KUKA KRL program: MyProgram_156().src

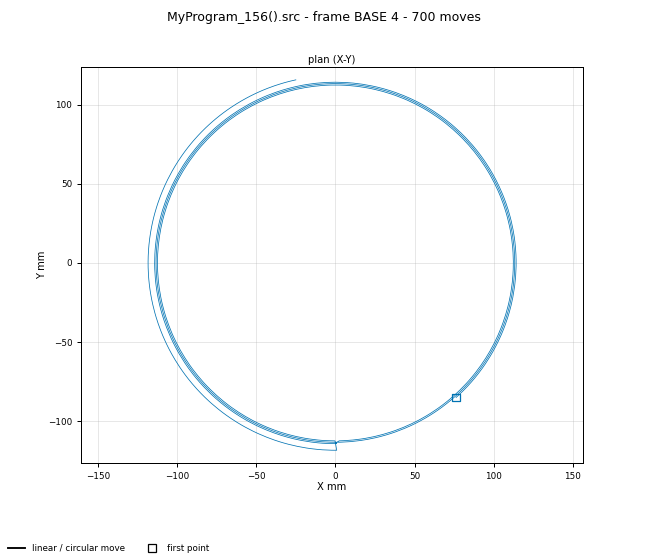
[picture p0: tool path of MyProgram_156().src in frame BASE 4, 700 of 700 moves have a stored position in this frame; points joined in program order, loops and branches not executed]
&ACCESS RVP
&REL 1
&PARAM TEMPLATE = C:\KRC\Roboter\Template\vorgabe
&PARAM EDITMASK = *
DEF MyProgram_156()
; ---- Setting reference (Base) ----
$BASE = BASE_DATA[4]

; --------------------------
; ---- Setting tool (TCP) ----
$TOOL = TOOL_DATA[3]
; --------------------------

$VEL.CP = VEL_APROX_PRINT
Startdeposition()
$VEL.CP = VEL_PRINT
LIN {X 76.2386,Y -85.0101,Z 120,A -51.5636,B 24.9513,C -1.613,E1 25.1077,E2 497.4724} C_DIS
LIN {X 78.7436,Y -82.698,Z 120,A -49.7889,B 24.9508,C -1.62,E1 25.1113,E2 495.6883} C_DIS
LIN {X 81.111,Y -80.3746,Z 120,A -48.1831,B 24.9508,C -1.6214,E1 25.1145,E2 494.086} C_DIS
LIN {X 83.3375,Y -78.0638,Z 120,A -46.5882,B 24.9505,C -1.6248,E1 25.1176,E2 492.4901} C_DIS
LIN {X 85.7956,Y -75.3542,Z 120,A -44.7139,B 24.9501,C -1.6313,E1 25.1211,E2 490.6088} C_DIS
LIN {X 88.0102,Y -72.7553,Z 120,A -42.9236,B 24.9496,C -1.6394,E1 25.1243,E2 488.8074} C_DIS
LIN {X 90.5109,Y -69.6191,Z 120,A -41.0242,B 24.9496,C -1.6396,E1 25.1275,E2 486.9167} C_DIS
LIN {X 92.7013,Y -66.6761,Z 120,A -39.1167,B 24.9491,C -1.6478,E1 25.1307,E2 484.999} C_DIS
LIN {X 94.7109,Y -63.7885,Z 120,A -37.4463,B 24.9491,C -1.6483,E1 25.1333,E2 483.3356} C_DIS
LIN {X 97.8312,Y -58.8925,Z 120,A -34.6127,B 24.9488,C -1.6529,E1 25.1375,E2 480.5054} C_DIS
LIN {X 99.5347,Y -55.9643,Z 120,A -32.8334,B 24.9483,C -1.6617,E1 25.14,E2 478.7147} C_DIS
LIN {X 101.2424,Y -52.813,Z 120,A -31.0463,B 24.948,C -1.6665,E1 25.1423,E2 476.9256} C_DIS
LIN {X 102.9812,Y -49.3349,Z 120,A -29.0203,B 24.9474,C -1.6759,E1 25.1448,E2 474.8882} C_DIS
LIN {X 104.7978,Y -45.3494,Z 120,A -26.7386,B 24.9467,C -1.6866,E1 25.1474,E2 472.5937} C_DIS
LIN {X 106.0833,Y -42.2573,Z 120,A -25.2084,B 24.9468,C -1.6848,E1 25.149,E2 471.0764} C_DIS
LIN {X 107.2709,Y -39.1408,Z 120,A -23.3343,B 24.9459,C -1.6995,E1 25.1509,E2 469.178} C_DIS
LIN {X 108.7458,Y -34.8355,Z 120,A -21.3851,B 24.9464,C -1.6909,E1 25.1525,E2 467.26} C_DIS
LIN {X 109.8552,Y -31.1591,Z 120,A -19.3865,B 24.9458,C -1.7005,E1 25.1541,E2 465.2504} C_DIS
LIN {X 111.0251,Y -26.6948,Z 120,A -17.1795,B 24.9457,C -1.7028,E1 25.1556,E2 463.0507} C_DIS
LIN {X 112.0611,Y -21.9428,Z 120,A -14.7665,B 24.9452,C -1.7094,E1 25.157,E2 460.6362} C_DIS
LIN {X 113.2585,Y -14.5453,Z 120,A -11.4137,B 24.9457,C -1.7024,E1 25.1585,E2 457.3196} C_DIS
LIN {X 113.8562,Y -8.7156,Z 120,A -7.9945,B 24.9436,C -1.7344,E1 25.1594,E2 453.8452} C_DIS
LIN {X 114.1732,Y -1.8883,Z 120,A -4.1574,B 24.9416,C -1.7648,E1 25.1598,E2 449.9591} C_DIS
LIN {X 114.1717,Y 1.9674,Z 120,A -2.7839,B 24.943,C -1.7446,E1 25.1598,E2 448.6415} C_DIS
LIN {X 114.0675,Y 5.2703,Z 120,A -0.544,B 24.9408,C -1.7775,E1 25.1595,E2 446.3374} C_DIS
LIN {X 113.8093,Y 9.3025,Z 120,A 1.5121,B 24.9403,C -1.7854,E1 25.159,E2 444.2749} C_DIS
LIN {X 113.3833,Y 13.5398,Z 120,A 2.9581,B 24.942,C -1.7596,E1 25.1586,E2 442.8981} C_DIS
LIN {X 112.9985,Y 16.4475,Z 120,A 5.1558,B 24.9394,C -1.7986,E1 25.1576,E2 440.6215} C_DIS
LIN {X 112.2633,Y 20.8817,Z 120,A 6.6108,B 24.9414,C -1.768,E1 25.157,E2 439.2473} C_DIS
LIN {X 111.1091,Y 26.3486,Z 120,A 9.4907,B 24.9406,C -1.7803,E1 25.1553,E2 436.355} C_DIS
LIN {X 110.4068,Y 29.1515,Z 120,A 10.964,B 24.9402,C -1.7859,E1 25.1542,E2 434.877} C_DIS
LIN {X 109.1219,Y 33.6376,Z 120,A 13.3219,B 24.9397,C -1.7938,E1 25.1524,E2 432.5139} C_DIS
LIN {X 108.0151,Y 37.0421,Z 120,A 15.1558,B 24.9392,C -1.801,E1 25.1507,E2 430.6734} C_DIS
LIN {X 106.7656,Y 40.4989,Z 120,A 16.8898,B 24.9392,C -1.8014,E1 25.149,E2 428.9482} C_DIS
LIN {X 105.6594,Y 43.3037,Z 120,A 18.5007,B 24.9386,C -1.8104,E1 25.1473,E2 427.3249} C_DIS
LIN {X 103.451,Y 48.3421,Z 120,A 21.0822,B 24.9386,C -1.81,E1 25.1444,E2 424.7583} C_DIS
LIN {X 101.3471,Y 52.6143,Z 120,A 23.6617,B 24.9375,C -1.8255,E1 25.1412,E2 422.156} C_DIS
LIN {X 99.5345,Y 55.9646,Z 120,A 25.5138,B 24.9374,C -1.8281,E1 25.1387,E2 420.3076} C_DIS
LIN {X 97.6359,Y 59.2139,Z 120,A 27.3716,B 24.9371,C -1.8317,E1 25.136,E2 418.4507} C_DIS
LIN {X 95.1175,Y 63.1811,Z 120,A 29.4198,B 24.9377,C -1.8236,E1 25.133,E2 416.4319} C_DIS
LIN {X 93.6732,Y 65.3024,Z 120,A 30.9566,B 24.9366,C -1.8384,E1 25.1305,E2 414.8677} C_DIS
LIN {X 91.5095,Y 68.302,Z 120,A 32.8457,B 24.9362,C -1.8446,E1 25.1273,E2 412.9732} C_DIS
LIN {X 89.4167,Y 71.0195,Z 120,A 35.121,B 24.9341,C -1.8744,E1 25.1233,E2 410.6381} C_DIS
LIN {X 86.5957,Y 74.4344,Z 120,A 36.6899,B 24.9359,C -1.8494,E1 25.1206,E2 409.1353} C_DIS
LIN {X 82.3085,Y 79.1477,Z 120,A 39.5817,B 24.9364,C -1.8427,E1 25.1152,E2 406.2722} C_DIS
LIN {X 79.422,Y 82.0442,Z 120,A 41.9376,B 24.9351,C -1.8609,E1 25.1104,E2 403.8831} C_DIS
LIN {X 75.0439,Y 86.0666,Z 120,A 44.8129,B 24.9351,C -1.8621,E1 25.1045,E2 401.0167} C_DIS
LIN {X 72.8834,Y 87.9037,Z 120,A 46.8965,B 24.9327,C -1.8949,E1 25.0999,E2 398.8635} C_DIS
LIN {X 69.624,Y 90.5071,Z 120,A 48.4215,B 24.9342,C -1.8729,E1 25.0967,E2 397.3962} C_DIS
LIN {X 66.4308,Y 92.8763,Z 120,A 50.5415,B 24.9336,C -1.882,E1 25.0918,E2 395.2621} C_DIS
LIN {X 62.5852,Y 95.5104,Z 120,A 52.7023,B 24.9339,C -1.8778,E1 25.0869,E2 393.1184} C_DIS
LIN {X 60.3508,Y 96.9374,Z 120,A 54.0595,B 24.9337,C -1.8811,E1 25.0837,E2 391.7578} C_DIS
LIN {X 57.0857,Y 98.8955,Z 120,A 55.9041,B 24.9337,C -1.8811,E1 25.0792,E2 389.9191} C_DIS
LIN {X 54.6498,Y 100.2621,Z 120,A 57.4025,B 24.9332,C -1.8873,E1 25.0755,E2 388.4101} C_DIS
LIN {X 51.2738,Y 102.0315,Z 120,A 59.4609,B 24.9326,C -1.8963,E1 25.0704,E2 386.3362} C_DIS
LIN {X 47.3144,Y 103.9259,Z 120,A 61.617,B 24.9326,C -1.8969,E1 25.0649,E2 384.1842} C_DIS
LIN {X 43.2541,Y 105.6796,Z 120,A 63.9554,B 24.932,C -1.9046,E1 25.0589,E2 381.833} C_DIS
LIN {X 38.0509,Y 107.6626,Z 120,A 66.4845,B 24.9326,C -1.8955,E1 25.0523,E2 379.3308} C_DIS
LIN {X 34.5457,Y 108.8395,Z 120,A 68.6595,B 24.9315,C -1.9111,E1 25.0465,E2 377.123} C_DIS
LIN {X 30.7609,Y 109.968,Z 120,A 70.3134,B 24.9325,C -1.898,E1 25.0421,E2 375.5027} C_DIS
LIN {X 26.7576,Y 111.0098,Z 120,A 72.2957,B 24.9327,C -1.8952,E1 25.0368,E2 373.5301} C_DIS
LIN {X 23.2459,Y 111.7978,Z 120,A 74.2356,B 24.9322,C -1.902,E1 25.0314,E2 371.5767} C_DIS
LIN {X 16.9448,Y 112.9255,Z 120,A 77.3058,B 24.9325,C -1.8969,E1 25.023,E2 368.5218} C_DIS
LIN {X 11.441,Y 113.6149,Z 120,A 80.939,B 24.9298,C -1.9344,E1 25.0127,E2 364.8022} C_DIS
LIN {X 6.4298,Y 114.0075,Z 120,A 82.3847,B 24.9332,C -1.8877,E1 25.009,E2 363.4678} C_DIS
LIN {X 0.0192,Y 114.1907,Z 120,A 85.9521,B 24.9322,C -1.9022,E1 24.999,E2 359.8666} C_DIS
LIN {X -5.4539,Y 114.0596,Z 120,A 88.5974,B 24.9325,C -1.897,E1 24.9916,E2 357.2332} C_DIS
LIN {X -12.2551,Y 113.5297,Z 120,A 91.9236,B 24.9329,C -1.8913,E1 24.9824,E2 353.9192} C_DIS
LIN {X -17.9444,Y 112.771,Z 120,A 94.876,B 24.9329,C -1.8924,E1 24.9742,E2 350.9618} C_DIS
LIN {X -21.0211,Y 112.2385,Z 120,A 97.068,B 24.931,C -1.9178,E1 24.968,E2 348.7072} C_DIS
LIN {X -24.9456,Y 111.4323,Z 120,A 98.8245,B 24.932,C -1.9052,E1 24.9633,E2 346.9784} C_DIS
LIN {X -29.9895,Y 110.1804,Z 120,A 101.1547,B 24.933,C -1.8909,E1 24.9571,E2 344.6789} C_DIS
LIN {X -33.4559,Y 109.1782,Z 120,A 103.0604,B 24.9328,C -1.8928,E1 24.9519,E2 342.7653} C_DIS
LIN {X -37.39,Y 107.8945,Z 120,A 105.1169,B 24.9331,C -1.8895,E1 24.9465,E2 340.713} C_DIS
LIN {X -42.6939,Y 105.9076,Z 120,A 108.1852,B 24.9327,C -1.8951,E1 24.9385,E2 337.6247} C_DIS
LIN {X -46.0433,Y 104.4952,Z 120,A 110.2515,B 24.9321,C -1.9025,E1 24.9331,E2 335.5359} C_DIS
LIN {X -49.5357,Y 102.8847,Z 120,A 111.373,B 24.9347,C -1.8658,E1 24.9305,E2 334.4987} C_DIS
LIN {X -51.8511,Y 101.7375,Z 120,A 112.8876,B 24.9343,C -1.8727,E1 24.9267,E2 332.9637} C_DIS
LIN {X -54.8258,Y 100.1667,Z 120,A 114.7339,B 24.934,C -1.8764,E1 24.9221,E2 331.1036} C_DIS
LIN {X -60.8098,Y 96.6506,Z 120,A 118.4997,B 24.9336,C -1.8816,E1 24.913,E2 327.3137} C_DIS
LIN {X -65.554,Y 93.4983,Z 120,A 121.5436,B 24.9335,C -1.8836,E1 24.906,E2 324.2548} C_DIS
LIN {X -68.6343,Y 91.26,Z 120,A 122.9574,B 24.9352,C -1.8591,E1 24.903,E2 322.8943} C_DIS
LIN {X -71.6379,Y 88.9222,Z 120,A 124.9947,B 24.9352,C -1.8602,E1 24.8985,E2 320.8468} C_DIS
LIN {X -74.5863,Y 86.4663,Z 120,A 126.8349,B 24.9357,C -1.8523,E1 24.8946,E2 319.0183} C_DIS
LIN {X -77.1405,Y 84.1926,Z 120,A 128.5557,B 24.9359,C -1.8486,E1 24.891,E2 317.2995} C_DIS
LIN {X -79.9011,Y 81.5787,Z 120,A 130.5038,B 24.9361,C -1.8456,E1 24.8871,E2 315.3503} C_DIS
LIN {X -82.3085,Y 79.1477,Z 120,A 132.1826,B 24.9365,C -1.8399,E1 24.8838,E2 313.678} C_DIS
LIN {X -85.738,Y 75.4202,Z 120,A 134.871,B 24.9365,C -1.8393,E1 24.8788,E2 310.9789} C_DIS
LIN {X -87.8307,Y 72.9712,Z 120,A 136.3419,B 24.9373,C -1.8292,E1 24.8762,E2 309.5253} C_DIS
LIN {X -92.1157,Y 67.4814,Z 120,A 139.6684,B 24.9384,C -1.813,E1 24.8706,E2 306.2217} C_DIS
LIN {X -94.7744,Y 63.6947,Z 120,A 142.1042,B 24.9385,C -1.8111,E1 24.8667,E2 303.7785} C_DIS
LIN {X -96.2133,Y 61.4987,Z 120,A 143.4703,B 24.9386,C -1.8093,E1 24.8646,E2 302.4098} C_DIS
LIN {X -99.3647,Y 56.2686,Z 120,A 146.8399,B 24.9384,C -1.8126,E1 24.8598,E2 299.0147} C_DIS
LIN {X -101.3602,Y 52.5893,Z 120,A 148.7275,B 24.9394,C -1.7978,E1 24.8573,E2 297.1523} C_DIS
LIN {X -103.3993,Y 48.4532,Z 120,A 151.1537,B 24.9396,C -1.7954,E1 24.8544,E2 294.7189} C_DIS
LIN {X -106.1097,Y 42.19,Z 120,A 154.3823,B 24.9408,C -1.777,E1 24.8509,E2 291.5163} C_DIS
LIN {X -107.202,Y 39.3297,Z 120,A 157.0353,B 24.9381,C -1.8172,E1 24.8483,E2 288.7523} C_DIS
LIN {X -109.0942,Y 33.727,Z 120,A 158.6626,B 24.9423,C -1.7539,E1 24.847,E2 287.2666} C_DIS
LIN {X -109.8654,Y 31.1231,Z 120,A 160.3997,B 24.9416,C -1.7645,E1 24.8456,E2 285.4943} C_DIS
LIN {X -111.222,Y 25.8599,Z 120,A 162.8599,B 24.9429,C -1.7451,E1 24.8439,E2 283.0659} C_DIS
LIN {X -111.7459,Y 23.4986,Z 120,A 164.4267,B 24.9423,C -1.7552,E1 24.843,E2 281.4659} C_DIS
LIN {X -112.3914,Y 20.1798,Z 120,A 166.0871,B 24.9427,C -1.7483,E1 24.8421,E2 279.812} C_DIS
LIN {X -113.0751,Y 15.9085,Z 120,A 168.2456,B 24.9432,C -1.7408,E1 24.8412,E2 277.6586} C_DIS
LIN {X -113.6182,Y 11.4094,Z 120,A 170.518,B 24.9437,C -1.7333,E1 24.8405,E2 275.3904} C_DIS
LIN {X -113.8778,Y 8.4455,Z 120,A 172.0471,B 24.9439,C -1.7299,E1 24.8401,E2 273.8604} C_DIS
LIN {X -114.0597,Y 5.4493,Z 120,A 173.7958,B 24.9436,C -1.7347,E1 24.8399,E2 272.0897} C_DIS
LIN {X -114.1877,Y -0.5465,Z 120,A 176.6355,B 24.9447,C -1.7181,E1 24.8399,E2 269.2724} C_DIS
LIN {X -114.1212,Y -3.9481,Z 120,A 178.4619,B 24.9447,C -1.7173,E1 24.8399,E2 267.4369} C_DIS
LIN {X -113.7849,Y -9.6066,Z 120,A -178.4365,B 24.9447,C -1.7185,E1 24.8406,E2 264.3139} C_DIS
LIN {X -113.4701,Y -12.7992,Z 120,A -177.3293,B 24.9463,C -1.6932,E1 24.8409,E2 263.2605} C_DIS
LIN {X -112.9768,Y -16.5995,Z 120,A -174.8603,B 24.9453,C -1.7089,E1 24.8419,E2 260.739} C_DIS
LIN {X -112.4554,Y -19.824,Z 120,A -173.585,B 24.9465,C -1.6891,E1 24.8425,E2 259.5035} C_DIS
LIN {X -111.8985,Y -22.7553,Z 120,A -172.0568,B 24.9468,C -1.6857,E1 24.8433,E2 257.9744} C_DIS
LIN {X -111.1311,Y -26.2534,Z 120,A -170.2104,B 24.947,C -1.682,E1 24.8444,E2 256.1259} C_DIS
LIN {X -110.272,Y -29.6503,Z 120,A -168.5105,B 24.9475,C -1.6743,E1 24.8456,E2 254.4346} C_DIS
LIN {X -109.3885,Y -32.761,Z 120,A -166.8336,B 24.9476,C -1.6715,E1 24.8469,E2 252.7546} C_DIS
LIN {X -108.25,Y -36.3455,Z 120,A -164.2457,B 24.9462,C -1.6942,E1 24.8493,E2 250.0977} C_DIS
LIN {X -106.6107,Y -40.9073,Z 120,A -162.5705,B 24.9486,C -1.6562,E1 24.8509,E2 248.5037} C_DIS
LIN {X -103.8533,Y -47.4753,Z 120,A -158.9719,B 24.9492,C -1.6467,E1 24.8548,E2 244.9078} C_DIS
LIN {X -102.3457,Y -50.6399,Z 120,A -157.1253,B 24.9492,C -1.6453,E1 24.8571,E2 243.0545} C_DIS
LIN {X -100.6772,Y -53.8846,Z 120,A -155.022,B 24.9489,C -1.6513,E1 24.8598,E2 240.9258} C_DIS
LIN {X -98.6721,Y -57.4745,Z 120,A -153.1831,B 24.9498,C -1.6366,E1 24.8624,E2 239.1125} C_DIS
LIN {X -95.0936,Y -63.2174,Z 120,A -149.9823,B 24.9508,C -1.6197,E1 24.8671,E2 235.9356} C_DIS
LIN {X -92.8073,Y -66.5275,Z 120,A -147.8552,B 24.9508,C -1.619,E1 24.8705,E2 233.7997} C_DIS
LIN {X -89.9271,Y -70.3736,Z 120,A -145.4098,B 24.9512,C -1.6144,E1 24.8746,E2 231.3534} C_DIS
LIN {X -87.8624,Y -72.9331,Z 120,A -143.7453,B 24.9514,C -1.6111,E1 24.8776,E2 229.6891} C_DIS
LIN {X -85.7278,Y -75.4319,Z 120,A -141.86,B 24.951,C -1.6171,E1 24.8811,E2 227.7812} C_DIS
LIN {X -82.7328,Y -78.7067,Z 120,A -139.6862,B 24.9514,C -1.6099,E1 24.8852,E2 225.6149} C_DIS
LIN {X -78.5953,Y -82.8376,Z 120,A -137.0135,B 24.9525,C -1.5929,E1 24.8905,E2 222.9715} C_DIS
LIN {X -75.4162,Y -85.7414,Z 120,A -134.6481,B 24.9522,C -1.597,E1 24.8954,E2 220.5867} C_DIS
LIN {X -72.2085,Y -88.4598,Z 120,A -132.6218,B 24.9527,C -1.5895,E1 24.8997,E2 218.5706} C_DIS
LIN {X -69.7896,Y -90.3796,Z 120,A -130.9737,B 24.9526,C -1.5908,E1 24.9034,E2 216.9133} C_DIS
LIN {X -66.8325,Y -92.5897,Z 120,A -129.0989,B 24.9527,C -1.5885,E1 24.9076,E2 215.0374} C_DIS
LIN {X -63.6085,Y -94.8328,Z 120,A -127.1457,B 24.953,C -1.5845,E1 24.9121,E2 213.0871} C_DIS
LIN {X -59.7782,Y -97.2921,Z 120,A -124.5248,B 24.9523,C -1.5953,E1 24.9184,E2 210.4323} C_DIS
LIN {X -57.0074,Y -98.9404,Z 120,A -123.3308,B 24.9535,C -1.575,E1 24.9212,E2 209.2829} C_DIS
LIN {X -54.373,Y -100.4123,Z 120,A -121.6249,B 24.9532,C -1.5811,E1 24.9254,E2 207.5577} C_DIS
LIN {X -50.3798,Y -102.4747,Z 120,A -119.524,B 24.9537,C -1.5717,E1 24.9306,E2 205.4736} C_DIS
LIN {X -48.1213,Y -103.5538,Z 120,A -118.2046,B 24.9537,C -1.5729,E1 24.9339,E2 204.148} C_DIS
LIN {X -43.8969,Y -105.4151,Z 120,A -115.5924,B 24.953,C -1.583,E1 24.9407,E2 201.5055} C_DIS
LIN {X -39.103,Y -107.2847,Z 120,A -113.2857,B 24.9539,C -1.5688,E1 24.9467,E2 199.2278} C_DIS
LIN {X -34.3136,Y -108.9123,Z 120,A -110.9186,B 24.9544,C -1.5594,E1 24.9529,E2 196.8787} C_DIS
LIN {X -30.0803,Y -110.1559,Z 120,A -108.525,B 24.9541,C -1.5657,E1 24.9594,E2 194.4664} C_DIS
LIN {X -26.125,Y -111.1607,Z 120,A -106.4824,B 24.9541,C -1.5643,E1 24.9649,E2 192.4242} C_DIS
LIN {X -21.571,Y -112.1327,Z 120,A -104.1706,B 24.9543,C -1.5622,E1 24.9712,E2 190.1146} C_DIS
LIN {X -15.0454,Y -113.1937,Z 120,A -100.3366,B 24.953,C -1.584,E1 24.982,E2 186.2258} C_DIS
LIN {X -11.092,Y -113.6502,Z 120,A -98.9589,B 24.9546,C -1.5565,E1 24.9856,E2 184.9123} C_DIS
LIN {X -8.1981,Y -113.895,Z 120,A -96.7306,B 24.9526,C -1.5905,E1 24.9921,E2 182.6025} C_DIS
LIN {X -3.6609,Y -114.13,Z 120,A -94.4111,B 24.9525,C -1.5926,E1 24.9985,E2 180.2778} C_DIS
LIN {X 0.826,Y -114.1802,Z 120,A -94.2003,B 24.9576,C -1.5037,E1 24.9986,E2 180.2778} C_DIS
Enddeposition()
LIN {X 0.826,Y -114.1802,Z 120,A -94.2003,B 24.9576,C -1.5037,E1 24.9986,E2 180.2778} C_DIS
Startdeposition()
$VEL.CP = VEL_PRINT
LIN {X 0.5604,Y -113.3011,Z 120,A -94.2192,B 24.9565,C -1.5242,E1 24.9986,E2 180.248} C_DIS
LIN {X -3.0264,Y -113.2628,Z 120,A -96.4904,B 24.9576,C -1.5045,E1 24.9922,E2 182.5661} C_DIS
LIN {X -8.552,Y -112.9802,Z 120,A -98.2379,B 24.955,C -1.5491,E1 24.9876,E2 184.2085} C_DIS
LIN {X -14.2204,Y -112.407,Z 120,A -101.0574,B 24.9549,C -1.552,E1 24.9798,E2 187.0228} C_DIS
LIN {X -17.25,Y -111.9816,Z 120,A -102.8667,B 24.9555,C -1.5412,E1 24.9747,E2 188.8592} C_DIS
LIN {X -20.5468,Y -111.4249,Z 120,A -104.7709,B 24.956,C -1.5328,E1 24.9694,E2 190.7855} C_DIS
LIN {X -25.1163,Y -110.4842,Z 120,A -106.6838,B 24.9548,C -1.5527,E1 24.9643,E2 192.6533} C_DIS
LIN {X -27.1879,Y -109.9926,Z 120,A -108.0573,B 24.9555,C -1.5408,E1 24.9605,E2 194.0571} C_DIS
LIN {X -30.4687,Y -109.1296,Z 120,A -109.4981,B 24.9548,C -1.5534,E1 24.9567,E2 195.4701} C_DIS
LIN {X -32.6296,Y -108.5031,Z 120,A -110.7626,B 24.9551,C -1.5489,E1 24.9532,E2 196.7475} C_DIS
LIN {X -36.2392,Y -107.3506,Z 120,A -112.7597,B 24.9551,C -1.547,E1 24.9479,E2 198.7526} C_DIS
LIN {X -40.1007,Y -105.9687,Z 120,A -115.9071,B 24.9576,C -1.5046,E1 24.9394,E2 202.0074} C_DIS
LIN {X -46.0582,Y -103.5199,Z 120,A -117.9469,B 24.9545,C -1.5582,E1 24.9345,E2 203.9245} C_DIS
LIN {X -49.2376,Y -102.0447,Z 120,A -119.94,B 24.9549,C -1.5511,E1 24.9294,E2 205.9395} C_DIS
LIN {X -52.2376,Y -100.5438,Z 120,A -121.7297,B 24.955,C -1.5494,E1 24.9249,E2 207.7381} C_DIS
LIN {X -56.2111,Y -98.3759,Z 120,A -125.0629,B 24.9573,C -1.5102,E1 24.9166,E2 211.1743} C_DIS
LIN {X -62.0967,Y -94.7709,Z 120,A -127.6485,B 24.9549,C -1.5522,E1 24.9108,E2 213.6683} C_DIS
LIN {X -65.4261,Y -92.5044,Z 120,A -129.2346,B 24.9536,C -1.574,E1 24.9072,E2 215.2079} C_DIS
LIN {X -67.4604,Y -91.0326,Z 120,A -130.8072,B 24.9542,C -1.5639,E1 24.9036,E2 216.8103} C_DIS
LIN {X -70.3716,Y -88.7991,Z 120,A -132.4081,B 24.9534,C -1.5776,E1 24.9001,E2 218.3844} C_DIS
LIN {X -72.4498,Y -87.1118,Z 120,A -133.9467,B 24.9537,C -1.5727,E1 24.8968,E2 219.9406} C_DIS
LIN {X -75.6065,Y -84.3865,Z 120,A -136.0737,B 24.9535,C -1.5761,E1 24.8923,E2 222.0677} C_DIS
LIN {X -79.0329,Y -81.1884,Z 120,A -138.5976,B 24.9535,C -1.5748,E1 24.8872,E2 224.6052} C_DIS
LIN {X -82.1695,Y -78.0121,Z 120,A -140.6064,B 24.9526,C -1.5897,E1 24.8833,E2 226.587} C_DIS
LIN {X -84.1808,Y -75.8363,Z 120,A -142.2397,B 24.9528,C -1.5877,E1 24.8802,E2 228.2325} C_DIS
LIN {X -86.4828,Y -73.2003,Z 120,A -144.0611,B 24.9526,C -1.5897,E1 24.8769,E2 230.0573} C_DIS
LIN {X -88.8268,Y -70.3366,Z 120,A -145.8907,B 24.9523,C -1.5959,E1 24.8737,E2 231.8808} C_DIS
LIN {X -91.1598,Y -67.2868,Z 120,A -147.7112,B 24.9517,C -1.6055,E1 24.8707,E2 233.6871} C_DIS
LIN {X -92.9577,Y -64.7789,Z 120,A -149.2891,B 24.9515,C -1.6088,E1 24.8681,E2 235.265} C_DIS
LIN {X -94.2783,Y -62.8439,Z 120,A -151.1301,B 24.9529,C -1.5858,E1 24.8652,E2 237.1699} C_DIS
LIN {X -96.5397,Y -59.3112,Z 120,A -152.7773,B 24.9514,C -1.6101,E1 24.8629,E2 238.7677} C_DIS
LIN {X -97.9455,Y -56.9602,Z 120,A -154.4851,B 24.952,C -1.6011,E1 24.8604,E2 240.5058} C_DIS
LIN {X -99.5879,Y -54.034,Z 120,A -155.8188,B 24.9508,C -1.6201,E1 24.8587,E2 241.8013} C_DIS
LIN {X -101.1826,Y -50.9895,Z 120,A -157.5902,B 24.9506,C -1.6236,E1 24.8564,E2 243.5738} C_DIS
LIN {X -102.5679,Y -48.1393,Z 120,A -158.9446,B 24.9497,C -1.638,E1 24.8548,E2 244.9012} C_DIS
LIN {X -104.4003,Y -44.0227,Z 120,A -161.4285,B 24.9498,C -1.6364,E1 24.852,E2 247.4024} C_DIS
LIN {X -105.7208,Y -40.7553,Z 120,A -163.1504,B 24.9494,C -1.644,E1 24.8502,E2 249.1159} C_DIS
LIN {X -107.2805,Y -36.4471,Z 120,A -165.3923,B 24.9487,C -1.6539,E1 24.8482,E2 251.3469} C_DIS
LIN {X -107.9978,Y -34.2683,Z 120,A -166.8507,B 24.9493,C -1.6457,E1 24.8469,E2 252.8334} C_DIS
LIN {X -109.0319,Y -30.8136,Z 120,A -168.5498,B 24.9486,C -1.6562,E1 24.8456,E2 254.5172} C_DIS
LIN {X -109.9863,Y -27.2134,Z 120,A -170.2804,B 24.9479,C -1.668,E1 24.8444,E2 256.2298} C_DIS
LIN {X -110.5155,Y -24.9808,Z 120,A -171.7509,B 24.9484,C -1.6594,E1 24.8434,E2 257.7293} C_DIS
LIN {X -111.2888,Y -21.2665,Z 120,A -173.5467,B 24.9477,C -1.6703,E1 24.8424,E2 259.5098} C_DIS
LIN {X -111.883,Y -17.8876,Z 120,A -175.4201,B 24.9477,C -1.6703,E1 24.8416,E2 261.3942} C_DIS
LIN {X -112.4605,Y -13.8002,Z 120,A -177.5051,B 24.9473,C -1.6771,E1 24.8408,E2 263.4756} C_DIS
LIN {X -112.8326,Y -10.3075,Z 120,A -179.2013,B 24.9467,C -1.686,E1 24.8404,E2 265.1608} C_DIS
LIN {X -113.1095,Y -6.618,Z 120,A 179.1384,B 24.9458,C -1.7002,E1 24.84,E2 266.7971} C_DIS
LIN {X -113.247,Y -3.543,Z 120,A 177.6963,B 24.9452,C -1.7097,E1 24.8399,E2 268.2252} C_DIS
LIN {X -113.3003,Y -0.7681,Z 120,A 175.9113,B 24.9459,C -1.6994,E1 24.8398,E2 270.0456} C_DIS
LIN {X -113.2699,Y 2.7974,Z 120,A 174.1791,B 24.9453,C -1.708,E1 24.8398,E2 271.7677} C_DIS
LIN {X -113.1305,Y 6.2384,Z 120,A 172.3105,B 24.9453,C -1.7087,E1 24.8401,E2 273.6459} C_DIS
LIN {X -112.8168,Y 10.4788,Z 120,A 170.1496,B 24.9449,C -1.7153,E1 24.8406,E2 275.804} C_DIS
LIN {X -112.4248,Y 14.0825,Z 120,A 168.3044,B 24.9445,C -1.7208,E1 24.8412,E2 277.6472} C_DIS
LIN {X -111.9397,Y 17.5208,Z 120,A 166.5565,B 24.9441,C -1.7268,E1 24.8419,E2 279.3911} C_DIS
LIN {X -111.3768,Y 20.8095,Z 120,A 164.8263,B 24.9439,C -1.7306,E1 24.8428,E2 281.1226} C_DIS
LIN {X -110.7164,Y 24.0691,Z 120,A 163.1268,B 24.9436,C -1.7353,E1 24.8438,E2 282.8208} C_DIS
LIN {X -109.9826,Y 27.2287,Z 120,A 161.4836,B 24.9432,C -1.7405,E1 24.8448,E2 284.4613} C_DIS
LIN {X -109.0539,Y 30.736,Z 120,A 159.6851,B 24.9428,C -1.7477,E1 24.8461,E2 286.253} C_DIS
LIN {X -108.3381,Y 33.1728,Z 120,A 158.0515,B 24.9434,C -1.7383,E1 24.8475,E2 287.9186} C_DIS
LIN {X -106.831,Y 37.7443,Z 120,A 156.0026,B 24.9419,C -1.7609,E1 24.8493,E2 289.9253} C_DIS
LIN {X -105.7069,Y 40.7913,Z 120,A 154.2658,B 24.9418,C -1.7623,E1 24.851,E2 291.6686} C_DIS
LIN {X -104.4838,Y 43.8246,Z 120,A 152.4811,B 24.9418,C -1.7623,E1 24.8529,E2 293.4631} C_DIS
LIN {X -103.0723,Y 47.0513,Z 120,A 150.6971,B 24.9414,C -1.7676,E1 24.855,E2 295.2443} C_DIS
LIN {X -101.2371,Y 50.8809,Z 120,A 148.7442,B 24.9405,C -1.7816,E1 24.8573,E2 297.1742} C_DIS
LIN {X -98.9316,Y 55.2266,Z 120,A 146.2901,B 24.9399,C -1.7903,E1 24.8606,E2 299.6206} C_DIS
LIN {X -97.2506,Y 58.1383,Z 120,A 144.5048,B 24.9399,C -1.7919,E1 24.8631,E2 301.4115} C_DIS
LIN {X -95.4464,Y 61.0528,Z 120,A 142.9799,B 24.9389,C -1.8051,E1 24.8653,E2 302.9127} C_DIS
LIN {X -93.7931,Y 63.5632,Z 120,A 141.4771,B 24.9386,C -1.81,E1 24.8676,E2 304.4112} C_DIS
LIN {X -92.0085,Y 66.1211,Z 120,A 138.7674,B 24.9413,C -1.7701,E1 24.8722,E2 307.2292} C_DIS
LIN {X -88.8362,Y 70.3247,Z 120,A 136.8806,B 24.9388,C -1.8075,E1 24.8753,E2 309.0358} C_DIS
LIN {X -87.2193,Y 72.3204,Z 120,A 134.6491,B 24.941,C -1.7745,E1 24.8795,E2 311.3561} C_DIS
LIN {X -83.3552,Y 76.7422,Z 120,A 132.6535,B 24.9379,C -1.8201,E1 24.883,E2 313.252} C_DIS
LIN {X -80.9831,Y 79.243,Z 120,A 130.8101,B 24.9379,C -1.8205,E1 24.8866,E2 315.1026} C_DIS
LIN {X -78.498,Y 81.7039,Z 120,A 129.0384,B 24.9376,C -1.8246,E1 24.8901,E2 316.8717} C_DIS
LIN {X -75.7216,Y 84.2835,Z 120,A 127.1635,B 24.9372,C -1.8308,E1 24.894,E2 318.7397} C_DIS
LIN {X -71.4959,Y 87.8966,Z 120,A 124.3506,B 24.9367,C -1.837,E1 24.9,E2 321.5485} C_DIS
LIN {X -69.2532,Y 89.674,Z 120,A 122.1825,B 24.9385,C -1.8116,E1 24.905,E2 323.7851} C_DIS
LIN {X -65.3735,Y 92.542,Z 120,A 120.3391,B 24.9365,C -1.8402,E1 24.909,E2 325.5668} C_DIS
LIN {X -62.2386,Y 94.6774,Z 120,A 118.4668,B 24.9361,C -1.8458,E1 24.9133,E2 327.4319} C_DIS
LIN {X -59.3315,Y 96.5274,Z 120,A 116.8942,B 24.9354,C -1.8559,E1 24.917,E2 328.9855} C_DIS
LIN {X -56.5573,Y 98.177,Z 120,A 115.3408,B 24.935,C -1.8621,E1 24.9207,E2 330.5289} C_DIS
LIN {X -54.7472,Y 99.1993,Z 120,A 114.0842,B 24.9355,C -1.8556,E1 24.9238,E2 331.8045} C_DIS
LIN {X -51.81,Y 100.7632,Z 120,A 112.5543,B 24.9348,C -1.8646,E1 24.9276,E2 333.3172} C_DIS
LIN {X -49.6816,Y 101.8314,Z 120,A 111.2532,B 24.935,C -1.8626,E1 24.9308,E2 334.6265} C_DIS
LIN {X -47.0272,Y 103.0832,Z 120,A 109.6426,B 24.9352,C -1.8598,E1 24.9349,E2 336.2478} C_DIS
LIN {X -39.4582,Y 106.2117,Z 120,A 105.4481,B 24.9349,C -1.8634,E1 24.9458,E2 340.443} C_DIS
LIN {X -35.3941,Y 107.6335,Z 120,A 103.4893,B 24.9341,C -1.875,E1 24.9509,E2 342.3779} C_DIS
LIN {X -32.4048,Y 108.5697,Z 120,A 101.8356,B 24.9341,C -1.874,E1 24.9553,E2 344.0369} C_DIS
LIN {X -29.9852,Y 109.2635,Z 120,A 100.4488,B 24.9344,C -1.8707,E1 24.9591,E2 345.4338} C_DIS
LIN {X -24.1725,Y 110.6938,Z 120,A 97.469,B 24.9341,C -1.8755,E1 24.9672,E2 348.4062} C_DIS
LIN {X -20.8431,Y 111.3703,Z 120,A 95.6718,B 24.9341,C -1.8736,E1 24.9721,E2 350.2099} C_DIS
LIN {X -17.223,Y 111.9857,Z 120,A 93.6869,B 24.9345,C -1.8697,E1 24.9776,E2 352.2059} C_DIS
LIN {X -13.137,Y 112.5382,Z 120,A 92.0604,B 24.933,C -1.89,E1 24.982,E2 353.7855} C_DIS
LIN {X -9.4968,Y 112.9046,Z 120,A 89.7902,B 24.9342,C -1.8734,E1 24.9884,E2 356.0962} C_DIS
LIN {X -5.3758,Y 113.1759,Z 120,A 87.9936,B 24.9333,C -1.8863,E1 24.9933,E2 357.8625} C_DIS
LIN {X -1.9417,Y 113.2858,Z 120,A 85.9388,B 24.9342,C -1.8736,E1 24.9992,E2 359.948} C_DIS
LIN {X 2.8159,Y 113.2693,Z 120,A 83.6547,B 24.9338,C -1.879,E1 25.0055,E2 362.2188} C_DIS
LIN {X 6.0324,Y 113.1419,Z 120,A 81.6682,B 24.9349,C -1.864,E1 25.0111,E2 364.2402} C_DIS
LIN {X 9.4876,Y 112.9053,Z 120,A 80.0728,B 24.9344,C -1.8704,E1 25.0155,E2 365.8195} C_DIS
LIN {X 13.9176,Y 112.4462,Z 120,A 78.1496,B 24.9335,C -1.8839,E1 25.0208,E2 367.7094} C_DIS
LIN {X 16.6582,Y 112.0731,Z 120,A 76.7205,B 24.9335,C -1.8823,E1 25.0247,E2 369.1411} C_DIS
LIN {X 20.2987,Y 111.4695,Z 120,A 74.7508,B 24.9339,C -1.8772,E1 25.0302,E2 371.1207} C_DIS
LIN {X 23.2543,Y 110.8914,Z 120,A 73.3673,B 24.9336,C -1.8825,E1 25.0339,E2 372.4901} C_DIS
LIN {X 26.0046,Y 110.279,Z 120,A 71.8343,B 24.9339,C -1.8771,E1 25.0381,E2 374.0337} C_DIS
LIN {X 28.833,Y 109.5742,Z 120,A 70.4579,B 24.9337,C -1.8803,E1 25.0418,E2 375.4004} C_DIS
LIN {X 31.0593,Y 108.9623,Z 120,A 69.3581,B 24.9336,C -1.8825,E1 25.0448,E2 376.4933} C_DIS
LIN {X 33.5937,Y 108.2076,Z 120,A 67.8357,B 24.9342,C -1.8735,E1 25.0489,E2 378.0343} C_DIS
LIN {X 37.3046,Y 106.9852,Z 120,A 65.0288,B 24.9368,C -1.8362,E1 25.0565,E2 380.9238} C_DIS
LIN {X 42.4877,Y 105.0347,Z 120,A 63.1176,B 24.9343,C -1.8715,E1 25.0613,E2 382.7472} C_DIS
LIN {X 45.8341,Y 103.6197,Z 120,A 61.1747,B 24.9348,C -1.8649,E1 25.0663,E2 384.7012} C_DIS
LIN {X 49.3579,Y 101.9869,Z 120,A 59.2041,B 24.935,C -1.8622,E1 25.0712,E2 386.6729} C_DIS
LIN {X 52.8569,Y 100.2177,Z 120,A 57.3545,B 24.9348,C -1.8654,E1 25.0758,E2 388.5098} C_DIS
LIN {X 55.6354,Y 98.7033,Z 120,A 55.4893,B 24.9357,C -1.8516,E1 25.0804,E2 390.4022} C_DIS
LIN {X 59.8289,Y 96.2184,Z 120,A 53.2606,B 24.9353,C -1.8582,E1 25.0857,E2 392.6084} C_DIS
LIN {X 63.1587,Y 94.067,Z 120,A 51.482,B 24.9348,C -1.8649,E1 25.0898,E2 394.3652} C_DIS
LIN {X 65.5829,Y 92.3926,Z 120,A 49.7885,B 24.9356,C -1.8534,E1 25.0937,E2 396.0801} C_DIS
LIN {X 68.8412,Y 89.9915,Z 120,A 47.6174,B 24.9362,C -1.8442,E1 25.0986,E2 398.265} C_DIS
LIN {X 72.142,Y 87.3675,Z 120,A 45.6115,B 24.9362,C -1.8458,E1 25.1029,E2 400.2597} C_DIS
LIN {X 74.8577,Y 85.0526,Z 120,A 43.9915,B 24.9358,C -1.8504,E1 25.1063,E2 401.8624} C_DIS
LIN {X 77.0541,Y 83.0691,Z 120,A 42.332,B 24.9365,C -1.8401,E1 25.1097,E2 403.5396} C_DIS
LIN {X 79.532,Y 80.6976,Z 120,A 40.6274,B 24.9367,C -1.8378,E1 25.1132,E2 405.2426} C_DIS
LIN {X 81.3864,Y 78.8273,Z 120,A 39.1968,B 24.9372,C -1.8304,E1 25.116,E2 406.6844} C_DIS
LIN {X 84.3127,Y 75.689,Z 120,A 37.1583,B 24.9372,C -1.8314,E1 25.1198,E2 408.7116} C_DIS
LIN {X 86.7423,Y 72.8944,Z 120,A 35.0635,B 24.9381,C -1.8171,E1 25.1236,E2 410.8308} C_DIS
LIN {X 89.7885,Y 69.1047,Z 120,A 32.8258,B 24.9378,C -1.821,E1 25.1275,E2 413.0486} C_DIS
LIN {X 91.8285,Y 66.3735,Z 120,A 31.0737,B 24.9382,C -1.8154,E1 25.1304,E2 414.8055} C_DIS
LIN {X 93.3892,Y 64.1582,Z 120,A 29.6522,B 24.9386,C -1.8096,E1 25.1327,E2 416.2337} C_DIS
LIN {X 95.0391,Y 61.6873,Z 120,A 28.2026,B 24.9387,C -1.808,E1 25.1349,E2 417.6797} C_DIS
LIN {X 96.8528,Y 58.796,Z 120,A 26.5912,B 24.9387,C -1.8087,E1 25.1372,E2 419.2815} C_DIS
LIN {X 98.67,Y 55.6949,Z 120,A 24.8093,B 24.9389,C -1.8053,E1 25.1397,E2 421.062} C_DIS
LIN {X 99.9936,Y 53.2823,Z 120,A 23.2783,B 24.9396,C -1.7951,E1 25.1417,E2 422.6091} C_DIS
LIN {X 101.6033,Y 50.1421,Z 120,A 21.6178,B 24.9396,C -1.7958,E1 25.1438,E2 424.2592} C_DIS
LIN {X 103.0486,Y 47.104,Z 120,A 19.694,B 24.9406,C -1.7808,E1 25.1461,E2 426.2081} C_DIS
LIN {X 104.8701,Y 42.892,Z 120,A 17.6221,B 24.9403,C -1.7853,E1 25.1483,E2 428.2578} C_DIS
LIN {X 105.9094,Y 40.2572,Z 120,A 16.3196,B 24.9401,C -1.787,E1 25.1496,E2 429.5491} C_DIS
LIN {X 106.7088,Y 38.0925,Z 120,A 15.1167,B 24.9405,C -1.7818,E1 25.1508,E2 430.7574} C_DIS
LIN {X 107.7211,Y 35.1234,Z 120,A 13.4363,B 24.9411,C -1.7728,E1 25.1523,E2 432.4497} C_DIS
LIN {X 108.8089,Y 31.5987,Z 120,A 11.425,B 24.9419,C -1.7604,E1 25.1539,E2 434.4789} C_DIS
LIN {X 109.9078,Y 27.535,Z 120,A 9.323,B 24.9423,C -1.755,E1 25.1554,E2 436.5814} C_DIS
LIN {X 110.8666,Y 23.3751,Z 120,A 7.2529,B 24.9425,C -1.7523,E1 25.1566,E2 438.6458} C_DIS
LIN {X 112.0003,Y 17.1287,Z 120,A 4.025,B 24.9432,C -1.7413,E1 25.1582,E2 441.8806} C_DIS
LIN {X 112.9074,Y 9.4628,Z 120,A -0.5243,B 24.9459,C -1.6993,E1 25.1595,E2 446.502} C_DIS
LIN {X 113.22,Y 4.3507,Z 120,A -2.2496,B 24.9439,C -1.7304,E1 25.1597,E2 448.1438} C_DIS
LIN {X 113.3022,Y 0.3158,Z 120,A -4.4655,B 24.9448,C -1.7157,E1 25.1597,E2 450.3811} C_DIS
LIN {X 113.2156,Y -4.426,Z 120,A -7.0756,B 24.946,C -1.6982,E1 25.1596,E2 453.017} C_DIS
LIN {X 113.0427,Y -7.6661,Z 120,A -8.4016,B 24.9454,C -1.7073,E1 25.1593,E2 454.3137} C_DIS
LIN {X 112.4375,Y -13.9845,Z 120,A -12.2421,B 24.9479,C -1.6679,E1 25.1581,E2 458.2242} C_DIS
LIN {X 111.7615,Y -18.6224,Z 120,A -13.9413,B 24.9464,C -1.691,E1 25.1574,E2 459.8592} C_DIS
LIN {X 111.2061,Y -21.6957,Z 120,A -15.6698,B 24.9472,C -1.679,E1 25.1565,E2 461.6059} C_DIS
LIN {X 110.2591,Y -26.0909,Z 120,A -17.8774,B 24.9474,C -1.6746,E1 25.1551,E2 463.8109} C_DIS
LIN {X 109.4464,Y -29.3084,Z 120,A -19.3868,B 24.9473,C -1.677,E1 25.1541,E2 465.3059} C_DIS
LIN {X 108.5351,Y -32.5217,Z 120,A -20.9582,B 24.9473,C -1.677,E1 25.1529,E2 466.8683} C_DIS
LIN {X 107.5356,Y -35.6906,Z 120,A -22.8284,B 24.9482,C -1.663,E1 25.1512,E2 468.761} C_DIS
LIN {X 106.135,Y -39.6615,Z 120,A -24.9089,B 24.9485,C -1.6586,E1 25.1493,E2 470.8404} C_DIS
LIN {X 105.0867,Y -42.36,Z 120,A -26.9479,B 24.9504,C -1.6277,E1 25.1471,E2 472.9408} C_DIS
LIN {X 103.3309,Y -46.4774,Z 120,A -28.2046,B 24.9479,C -1.6669,E1 25.1458,E2 474.0982} C_DIS
LIN {X 101.845,Y -49.6532,Z 120,A -30.4248,B 24.9495,C -1.6409,E1 25.1431,E2 476.3679} C_DIS
LIN {X 100.5143,Y -52.2936,Z 120,A -31.9101,B 24.9498,C -1.6368,E1 25.1411,E2 477.8548} C_DIS
LIN {X 98.6195,Y -55.7854,Z 120,A -33.8833,B 24.9501,C -1.6325,E1 25.1385,E2 479.8279} C_DIS
LIN {X 96.638,Y -59.1494,Z 120,A -36.1161,B 24.9511,C -1.615,E1 25.1352,E2 482.0906} C_DIS
LIN {X 94.877,Y -61.9359,Z 120,A -37.4811,B 24.9506,C -1.624,E1 25.1332,E2 483.4276} C_DIS
LIN {X 92.9544,Y -64.7837,Z 120,A -39.0701,B 24.9505,C -1.6259,E1 25.1307,E2 485.0042} C_DIS
LIN {X 90.967,Y -67.5487,Z 120,A -40.9651,B 24.9512,C -1.6132,E1 25.1275,E2 486.92} C_DIS
LIN {X 88.4428,Y -70.8219,Z 120,A -43.038,B 24.9515,C -1.6084,E1 25.1239,E2 488.9946} C_DIS
LIN {X 86.2625,Y -73.4589,Z 120,A -44.6369,B 24.9515,C -1.6098,E1 25.1211,E2 490.5829} C_DIS
LIN {X 84.029,Y -76.0059,Z 120,A -46.3879,B 24.9518,C -1.6036,E1 25.1178,E2 492.3405} C_DIS
LIN {X 81.6477,Y -78.5563,Z 120,A -48.1508,B 24.9521,C -1.5993,E1 25.1144,E2 494.1061} C_DIS
LIN {X 78.7974,Y -81.4154,Z 120,A -50.1451,B 24.9522,C -1.5964,E1 25.1105,E2 496.0988} C_DIS
LIN {X 76.429,Y -83.6426,Z 120,A -51.8313,B 24.9526,C -1.5906,E1 25.107,E2 497.7918} C_DIS
LIN {X 73.6162,Y -86.1285,Z 120,A -53.6759,B 24.9527,C -1.5886,E1 25.1031,E2 499.6339} C_DIS
LIN {X 70.8265,Y -88.4391,Z 120,A -55.6447,B 24.9533,C -1.5783,E1 25.0988,E2 501.6194} C_DIS
LIN {X 67.4866,Y -91.0135,Z 120,A -57.6926,B 24.9533,C -1.5775,E1 25.0943,E2 503.6618} C_DIS
LIN {X 65.085,Y -92.7449,Z 120,A -58.9488,B 24.9529,C -1.5853,E1 25.0915,E2 504.8953} C_DIS
LIN {X 62.4445,Y -94.5416,Z 120,A -60.6389,B 24.9533,C -1.5787,E1 25.0875,E2 506.5954} C_DIS
LIN {X 59.828,Y -96.219,Z 120,A -62.3025,B 24.9537,C -1.5715,E1 25.0836,E2 508.2706} C_DIS
LIN {X 56.9388,Y -97.9578,Z 120,A -63.8474,B 24.9535,C -1.5755,E1 25.0799,E2 509.8012} C_DIS
LIN {X 53.5144,Y -99.8697,Z 120,A -65.8837,B 24.9538,C -1.5696,E1 25.0749,E2 511.8456} C_DIS
LIN {X 50.785,Y -101.2847,Z 120,A -67.5519,B 24.9543,C -1.5619,E1 25.0707,E2 513.5273} C_DIS
LIN {X 47.566,Y -102.8347,Z 120,A -69.8764,B 24.9558,C -1.5362,E1 25.0647,E2 515.9069} C_DIS
LIN {X 43.7161,Y -104.5296,Z 120,A -71.5185,B 24.9547,C -1.5544,E1 25.0606,E2 517.502} C_DIS
LIN {X 40.2572,Y -105.9094,Z 120,A -73.1492,B 24.9542,C -1.5629,E1 25.0564,E2 519.1088} C_DIS
LIN {X 38.0925,Y -106.7088,Z 120,A -74.5609,B 24.955,C -1.5505,E1 25.0526,E2 520.547} C_DIS
LIN {X 34.8025,Y -107.825,Z 120,A -76.0428,B 24.9544,C -1.5605,E1 25.0488,E2 522.0024} C_DIS
LIN {X 31.8433,Y -108.7363,Z 120,A -77.733,B 24.9548,C -1.5532,E1 25.0442,E2 523.7069} C_DIS
LIN {X 28.2679,Y -109.7195,Z 120,A -79.7081,B 24.9552,C -1.5468,E1 25.0389,E2 525.694} C_DIS
LIN {X 25.126,Y -110.4819,Z 120,A -81.2737,B 24.9551,C -1.5483,E1 25.0346,E2 527.254} C_DIS
LIN {X 20.3647,Y -111.4576,Z 120,A -83.9861,B 24.9559,C -1.5351,E1 25.0271,E2 529.9944} C_DIS
LIN {X 15.9244,Y -112.1777,Z 120,A -85.7023,B 24.9545,C -1.5578,E1 25.0225,E2 531.6552} C_DIS
LIN {X 9.4896,Y -112.9052,Z 120,A -89.1004,B 24.955,C -1.5504,E1 25.0131,E2 535.0684} C_DIS
LIN {X 3.3835,Y -113.2519,Z 120,A -92.1276,B 24.9549,C -1.5519,E1 25.0047,E2 538.0909} C_DIS
LIN {X 0.8144,Y -113.2977,Z 120,A -92.9638,B 24.9537,C -1.5717,E1 25.0025,E2 538.8801} C_DIS
Enddeposition()
LIN {X 0.8144,Y -113.2977,Z 120,A -92.9638,B 24.9537,C -1.5717,E1 25.0025,E2 538.8801} C_DIS
Startdeposition()
$VEL.CP = VEL_PRINT
LIN {X 2.4378,Y -112.3903,Z 120,A -92.1544,B 24.9528,C -1.5865,E1 25.0048,E2 538.0358} C_DIS
LIN {X 5.49,Y -112.284,Z 120,A -90.6058,B 24.9528,C -1.5867,E1 25.0091,E2 536.4872} C_DIS
LIN {X 8.1952,Y -112.1187,Z 120,A -89.2283,B 24.9528,C -1.5871,E1 25.013,E2 535.1092} C_DIS
LIN {X 10.9817,Y -111.8804,Z 120,A -87.8023,B 24.9528,C -1.5879,E1 25.0169,E2 533.6822} C_DIS
LIN {X 13.6935,Y -111.5807,Z 120,A -86.4154,B 24.9528,C -1.5886,E1 25.0208,E2 532.2947} C_DIS
LIN {X 16.0578,Y -111.2636,Z 120,A -85.1532,B 24.9525,C -1.5915,E1 25.0243,E2 531.0268} C_DIS
LIN {X 19.1898,Y -110.7681,Z 120,A -83.5862,B 24.9525,C -1.5905,E1 25.0286,E2 529.4636} C_DIS
LIN {X 21.8757,Y -110.2689,Z 120,A -82.1967,B 24.9525,C -1.5916,E1 25.0324,E2 528.0732} C_DIS
LIN {X 24.5186,Y -109.7112,Z 120,A -80.824,B 24.9525,C -1.5927,E1 25.0361,E2 526.6997} C_DIS
LIN {X 27.2939,Y -109.0545,Z 120,A -79.3715,B 24.9524,C -1.5941,E1 25.0401,E2 525.246} C_DIS
LIN {X 29.9735,Y -108.3487,Z 120,A -77.9623,B 24.9524,C -1.5955,E1 25.0439,E2 523.8358} C_DIS
LIN {X 32.5986,Y -107.5878,Z 120,A -76.5727,B 24.9522,C -1.5969,E1 25.0476,E2 522.4453} C_DIS
LIN {X 35.066,Y -106.8082,Z 120,A -75.2734,B 24.9522,C -1.5977,E1 25.0511,E2 521.1465} C_DIS
LIN {X 37.8542,Y -105.8532,Z 120,A -73.7593,B 24.952,C -1.6001,E1 25.0551,E2 519.6297} C_DIS
LIN {X 40.4531,Y -104.8875,Z 120,A -72.3471,B 24.952,C -1.602,E1 25.0587,E2 518.2161} C_DIS
LIN {X 43.0001,Y -103.8692,Z 120,A -70.9568,B 24.9518,C -1.6037,E1 25.0623,E2 516.8249} C_DIS
LIN {X 45.475,Y -102.8094,Z 120,A -69.591,B 24.9518,C -1.6055,E1 25.0658,E2 515.4582} C_DIS
LIN {X 48.0474,Y -101.6331,Z 120,A -68.1521,B 24.9516,C -1.6077,E1 25.0695,E2 514.0179} C_DIS
LIN {X 50.5176,Y -100.4281,Z 120,A -66.7561,B 24.9514,C -1.6098,E1 25.073,E2 512.6207} C_DIS
LIN {X 52.9568,Y -99.1634,Z 120,A -65.3613,B 24.9514,C -1.6119,E1 25.0764,E2 511.2246} C_DIS
LIN {X 55.379,Y -97.8314,Z 120,A -63.9577,B 24.9512,C -1.6142,E1 25.0799,E2 509.8198} C_DIS
LIN {X 57.5035,Y -96.5963,Z 120,A -62.7354,B 24.9512,C -1.6152,E1 25.0828,E2 508.5988} C_DIS
LIN {X 60.1508,Y -94.9722,Z 120,A -61.136,B 24.9509,C -1.619,E1 25.0866,E2 506.9957} C_DIS
LIN {X 62.4435,Y -93.4808,Z 120,A -59.7451,B 24.9507,C -1.6216,E1 25.0898,E2 505.6032} C_DIS
LIN {X 64.7144,Y -91.9232,Z 120,A -58.3481,B 24.9506,C -1.6242,E1 25.0931,E2 504.2049} C_DIS
LIN {X 67.3106,Y -90.0374,Z 120,A -56.6539,B 24.9502,C -1.6303,E1 25.0969,E2 502.5022} C_DIS
LIN {X 69.8412,Y -88.0888,Z 120,A -55.0357,B 24.95,C -1.6334,E1 25.1004,E2 500.8826} C_DIS
LIN {X 72.3738,Y -86.0226,Z 120,A -53.4416,B 24.95,C -1.6339,E1 25.1039,E2 499.2935} C_DIS
LIN {X 74.4662,Y -84.2178,Z 120,A -52.0405,B 24.9498,C -1.6368,E1 25.1068,E2 497.891} C_DIS
LIN {X 76.2722,Y -82.5837,Z 120,A -50.7781,B 24.9496,C -1.6408,E1 25.1094,E2 496.6244} C_DIS
LIN {X 78.8755,Y -80.1004,Z 120,A -48.9376,B 24.9493,C -1.6455,E1 25.1131,E2 494.7804} C_DIS
LIN {X 80.934,Y -78.0197,Z 120,A -47.4957,B 24.9492,C -1.647,E1 25.1159,E2 493.3412} C_DIS
LIN {X 82.8281,Y -76.0059,Z 120,A -46.0965,B 24.949,C -1.6501,E1 25.1186,E2 491.9408} C_DIS
LIN {X 84.6596,Y -73.9604,Z 120,A -44.7267,B 24.9488,C -1.6524,E1 25.1211,E2 490.5717} C_DIS
LIN {X 86.5529,Y -71.7356,Z 120,A -43.1512,B 24.9483,C -1.6603,E1 25.124,E2 488.9848} C_DIS
LIN {X 88.6199,Y -69.1691,Z 120,A -41.5538,B 24.9483,C -1.661,E1 25.1267,E2 487.3932} C_DIS
LIN {X 90.2932,Y -66.9702,Z 120,A -40.1537,B 24.9481,C -1.6645,E1 25.1291,E2 485.9915} C_DIS
LIN {X 91.9064,Y -64.7385,Z 120,A -38.7585,B 24.9479,C -1.668,E1 25.1313,E2 484.5948} C_DIS
LIN {X 93.4538,Y -62.4836,Z 120,A -37.3786,B 24.9477,C -1.6713,E1 25.1335,E2 483.2139} C_DIS
LIN {X 94.9817,Y -60.1358,Z 120,A -35.9548,B 24.9474,C -1.6752,E1 25.1357,E2 481.7881} C_DIS
LIN {X 96.4349,Y -57.7767,Z 120,A -34.5602,B 24.9472,C -1.6785,E1 25.1377,E2 480.3928} C_DIS
LIN {X 97.8102,Y -55.4168,Z 120,A -33.1683,B 24.9469,C -1.6826,E1 25.1396,E2 478.9985} C_DIS
LIN {X 99.1454,Y -52.9911,Z 120,A -31.7664,B 24.9467,C -1.6864,E1 25.1415,E2 477.5951} C_DIS
LIN {X 100.4037,Y -50.5661,Z 120,A -30.3815,B 24.9465,C -1.6902,E1 25.1432,E2 476.2085} C_DIS
LIN {X 101.6106,Y -48.0948,Z 120,A -28.9939,B 24.9462,C -1.6938,E1 25.1449,E2 474.8198} C_DIS
LIN {X 102.7698,Y -45.5656,Z 120,A -27.5802,B 24.946,C -1.6979,E1 25.1465,E2 473.4041} C_DIS
LIN {X 103.7103,Y -43.3779,Z 120,A -26.3414,B 24.9457,C -1.7029,E1 25.1479,E2 472.1605} C_DIS
LIN {X 104.7112,Y -40.9024,Z 120,A -24.9677,B 24.9453,C -1.7077,E1 25.1493,E2 470.783} C_DIS
LIN {X 105.8462,Y -37.8741,Z 120,A -23.3793,B 24.9452,C -1.7101,E1 25.1508,E2 469.1978} C_DIS
LIN {X 106.7474,Y -35.2539,Z 120,A -21.9872,B 24.945,C -1.7136,E1 25.1521,E2 467.8053} C_DIS
LIN {X 107.5787,Y -32.6293,Z 120,A -20.5903,B 24.9447,C -1.7178,E1 25.1532,E2 466.4065} C_DIS
LIN {X 108.3405,Y -30.003,Z 120,A -19.2047,B 24.9444,C -1.7219,E1 25.1543,E2 465.0192} C_DIS
LIN {X 109.0427,Y -27.3409,Z 120,A -17.8111,B 24.9442,C -1.7259,E1 25.1553,E2 463.624} C_DIS
LIN {X 109.6794,Y -24.6627,Z 120,A -16.4177,B 24.9439,C -1.73,E1 25.1561,E2 462.2291} C_DIS
LIN {X 110.4311,Y -21.0334,Z 120,A -14.4886,B 24.9434,C -1.738,E1 25.1572,E2 460.2924} C_DIS
LIN {X 110.9847,Y -17.8943,Z 120,A -12.928,B 24.9432,C -1.7403,E1 25.1579,E2 458.7356} C_DIS
LIN {X 111.3901,Y -15.1673,Z 120,A -11.5328,B 24.943,C -1.7444,E1 25.1585,E2 457.3389} C_DIS
LIN {X 111.7314,Y -12.4072,Z 120,A -10.1253,B 24.9427,C -1.7486,E1 25.1589,E2 455.9299} C_DIS
LIN {X 111.9995,Y -9.691,Z 120,A -8.7485,B 24.9424,C -1.7524,E1 25.1593,E2 454.5522} C_DIS
LIN {X 112.1765,Y -7.3397,Z 120,A -7.5039,B 24.9421,C -1.7584,E1 25.1595,E2 453.301} C_DIS
LIN {X 112.3396,Y -4.1948,Z 120,A -5.9565,B 24.9419,C -1.7609,E1 25.1597,E2 451.7567} C_DIS
LIN {X 112.4083,Y -1.458,Z 120,A -4.5681,B 24.9416,C -1.7652,E1 25.1597,E2 450.3666} C_DIS
LIN {X 112.4122,Y 1.0357,Z 120,A -3.2862,B 24.9413,C -1.7698,E1 25.1597,E2 449.0814} C_DIS
LIN {X 112.3541,Y 3.7468,Z 120,A -1.912,B 24.941,C -1.7739,E1 25.1597,E2 447.7056} C_DIS
LIN {X 112.2312,Y 6.4504,Z 120,A -0.4903,B 24.9406,C -1.7804,E1 25.1594,E2 446.2771} C_DIS
LIN {X 111.9913,Y 9.7801,Z 120,A 1.097,B 24.9406,C -1.7806,E1 25.1591,E2 444.6989} C_DIS
LIN {X 111.7286,Y 12.431,Z 120,A 2.4586,B 24.9403,C -1.7851,E1 25.1587,E2 443.3346} C_DIS
LIN {X 111.4223,Y 14.923,Z 120,A 3.7529,B 24.94,C -1.7899,E1 25.1582,E2 442.0366} C_DIS
LIN {X 111.0012,Y 17.7908,Z 120,A 5.2097,B 24.9397,C -1.7937,E1 25.1576,E2 440.5795} C_DIS
LIN {X 110.5441,Y 20.4377,Z 120,A 6.5438,B 24.9395,C -1.7964,E1 25.157,E2 439.2468} C_DIS
LIN {X 109.9863,Y 23.256,Z 120,A 8.024,B 24.9392,C -1.8017,E1 25.1561,E2 437.7626} C_DIS
LIN {X 109.3753,Y 25.9788,Z 120,A 9.4353,B 24.9389,C -1.8057,E1 25.1552,E2 436.3503} C_DIS
LIN {X 108.7066,Y 28.6483,Z 120,A 10.83,B 24.9386,C -1.8097,E1 25.1543,E2 434.9542} C_DIS
LIN {X 107.9728,Y 31.3005,Z 120,A 12.2234,B 24.9384,C -1.8135,E1 25.1532,E2 433.5596} C_DIS
LIN {X 106.9181,Y 34.7263,Z 120,A 14.1123,B 24.9378,C -1.822,E1 25.1516,E2 431.6615} C_DIS
LIN {X 105.8532,Y 37.8542,Z 120,A 15.7119,B 24.9377,C -1.8231,E1 25.1501,E2 430.0682} C_DIS
LIN {X 104.8875,Y 40.4531,Z 120,A 17.116,B 24.9374,C -1.8269,E1 25.1488,E2 428.663} C_DIS
LIN {X 104.0711,Y 42.5043,Z 120,A 18.3085,B 24.937,C -1.8333,E1 25.1475,E2 427.462} C_DIS
LIN {X 102.7681,Y 45.5694,Z 120,A 19.9146,B 24.937,C -1.8341,E1 25.1457,E2 425.8629} C_DIS
LIN {X 101.6318,Y 48.0501,Z 120,A 21.3009,B 24.9367,C -1.8378,E1 25.1441,E2 424.4751} C_DIS
LIN {X 100.4272,Y 50.5193,Z 120,A 22.6951,B 24.9364,C -1.8415,E1 25.1423,E2 423.0798} C_DIS
LIN {X 99.1534,Y 52.9758,Z 120,A 24.0971,B 24.9362,C -1.8451,E1 25.1405,E2 421.6768} C_DIS
LIN {X 97.8159,Y 55.4068,Z 120,A 25.5029,B 24.9359,C -1.8486,E1 25.1386,E2 420.27} C_DIS
LIN {X 96.4294,Y 57.786,Z 120,A 26.8969,B 24.9357,C -1.8519,E1 25.1366,E2 418.8753} C_DIS
LIN {X 94.2267,Y 61.3122,Z 120,A 29.0013,B 24.9354,C -1.8568,E1 25.1335,E2 416.7699} C_DIS
LIN {X 92.6984,Y 63.5992,Z 120,A 30.3994,B 24.9351,C -1.8603,E1 25.1313,E2 415.3705} C_DIS
LIN {X 91.1255,Y 65.8329,Z 120,A 31.777,B 24.9349,C -1.8631,E1 25.129,E2 413.9929} C_DIS
LIN {X 89.4796,Y 68.0531,Z 120,A 33.1856,B 24.9347,C -1.8666,E1 25.1267,E2 412.5828} C_DIS
LIN {X 87.7786,Y 70.2336,Z 120,A 34.5878,B 24.9345,C -1.8697,E1 25.1243,E2 411.1799} C_DIS
LIN {X 86.0195,Y 72.3775,Z 120,A 35.9951,B 24.9343,C -1.8728,E1 25.1217,E2 409.7718} C_DIS
LIN {X 84.2193,Y 74.4645,Z 120,A 37.3918,B 24.934,C -1.8757,E1 25.1192,E2 408.3745} C_DIS
LIN {X 82.4038,Y 76.4683,Z 120,A 38.7639,B 24.9338,C -1.8786,E1 25.1166,E2 407.0018} C_DIS
LIN {X 80.4823,Y 78.4883,Z 120,A 40.3322,B 24.9332,C -1.8883,E1 25.1135,E2 405.4171} C_DIS
LIN {X 78.0211,Y 80.9327,Z 120,A 41.9391,B 24.9334,C -1.8849,E1 25.1103,E2 403.8251} C_DIS
LIN {X 76.0076,Y 82.8266,Z 120,A 43.3431,B 24.9332,C -1.8876,E1 25.1075,E2 402.4205} C_DIS
LIN {X 73.9522,Y 84.6668,Z 120,A 44.7392,B 24.933,C -1.8899,E1 25.1045,E2 401.0243} C_DIS
LIN {X 71.8514,Y 86.4567,Z 120,A 46.1399,B 24.9329,C -1.8924,E1 25.1015,E2 399.6232} C_DIS
LIN {X 69.7149,Y 88.1886,Z 120,A 47.5338,B 24.9327,C -1.8947,E1 25.0985,E2 398.2291} C_DIS
LIN {X 67.3125,Y 90.036,Z 120,A 49.0738,B 24.9325,C -1.8973,E1 25.0951,E2 396.6887} C_DIS
LIN {X 64.735,Y 91.9088,Z 120,A 50.6942,B 24.9323,C -1.8999,E1 25.0914,E2 395.0677} C_DIS
LIN {X 62.4738,Y 93.4604,Z 120,A 52.0865,B 24.9322,C -1.902,E1 25.0882,E2 393.6751} C_DIS
LIN {X 60.1673,Y 94.9617,Z 120,A 53.482,B 24.932,C -1.9039,E1 25.0849,E2 392.2796} C_DIS
LIN {X 57.9398,Y 96.336,Z 120,A 54.788,B 24.932,C -1.9047,E1 25.0818,E2 390.9758} C_DIS
LIN {X 55.4085,Y 97.8149,Z 120,A 56.3024,B 24.9318,C -1.9077,E1 25.0781,E2 389.4588} C_DIS
LIN {X 52.9959,Y 99.1428,Z 120,A 57.7026,B 24.9316,C -1.9095,E1 25.0747,E2 388.0584} C_DIS
LIN {X 50.5665,Y 100.4035,Z 120,A 59.0942,B 24.9316,C -1.9112,E1 25.0712,E2 386.6667} C_DIS
LIN {X 48.0832,Y 101.6161,Z 120,A 60.499,B 24.9314,C -1.9128,E1 25.0677,E2 385.2618} C_DIS
LIN {X 45.5654,Y 102.7699,Z 120,A 61.907,B 24.9314,C -1.9142,E1 25.0641,E2 383.8538} C_DIS
LIN {X 43.4925,Y 103.662,Z 120,A 63.1124,B 24.931,C -1.9179,E1 25.061,E2 382.6426} C_DIS
LIN {X 40.5534,Y 104.8482,Z 120,A 64.6647,B 24.9311,C -1.9168,E1 25.057,E2 381.0965} C_DIS
LIN {X 38.0851,Y 105.7692,Z 120,A 65.9964,B 24.9311,C -1.9176,E1 25.0535,E2 379.7656} C_DIS
LIN {X 35.3655,Y 106.7099,Z 120,A 67.4533,B 24.9311,C -1.9184,E1 25.0496,E2 378.3096} C_DIS
LIN {X 32.6409,Y 107.5752,Z 120,A 68.9249,B 24.9309,C -1.9201,E1 25.0457,E2 376.8366} C_DIS
LIN {X 29.9981,Y 108.3418,Z 120,A 70.3254,B 24.9309,C -1.921,E1 25.0419,E2 375.4363} C_DIS
LIN {X 27.3355,Y 109.044,Z 120,A 71.7271,B 24.9308,C -1.9218,E1 25.0381,E2 374.0348} C_DIS
LIN {X 24.6565,Y 109.6808,Z 120,A 73.1289,B 24.9308,C -1.9225,E1 25.0343,E2 372.6333} C_DIS
LIN {X 22.3482,Y 110.1727,Z 120,A 74.3748,B 24.9305,C -1.925,E1 25.0309,E2 371.3832} C_DIS
LIN {X 19.2293,Y 110.7614,Z 120,A 75.9464,B 24.9306,C -1.9236,E1 25.0266,E2 369.8166} C_DIS
LIN {X 16.4955,Y 111.2014,Z 120,A 77.3574,B 24.9306,C -1.924,E1 25.0227,E2 368.406} C_DIS
LIN {X 13.7946,Y 111.5685,Z 120,A 78.7461,B 24.9306,C -1.9243,E1 25.0189,E2 367.0177} C_DIS
LIN {X 11.05,Y 111.8737,Z 120,A 80.1528,B 24.9306,C -1.9245,E1 25.015,E2 365.6115} C_DIS
LIN {X 8.3396,Y 112.1081,Z 120,A 81.5395,B 24.9306,C -1.9245,E1 25.0111,E2 364.2253} C_DIS
LIN {X 5.9194,Y 112.2605,Z 120,A 82.8155,B 24.9304,C -1.9263,E1 25.0075,E2 362.9457} C_DIS
LIN {X 2.7776,Y 112.3838,Z 120,A 84.3782,B 24.9306,C -1.9244,E1 25.0032,E2 361.3878} C_DIS
LIN {X 0.0403,Y 112.418,Z 120,A 85.7737,B 24.9306,C -1.9242,E1 24.9993,E2 359.9929} C_DIS
LIN {X -2.6719,Y 112.386,Z 120,A 87.1567,B 24.9306,C -1.9239,E1 24.9954,E2 358.6107} C_DIS
LIN {X -5.1222,Y 112.2998,Z 120,A 88.448,B 24.9306,C -1.9252,E1 24.9918,E2 357.3158} C_DIS
LIN {X -8.1656,Y 112.1207,Z 120,A 89.9658,B 24.9306,C -1.923,E1 24.9876,E2 355.8026} C_DIS
LIN {X -10.9748,Y 111.881,Z 120,A 91.4014,B 24.9307,C -1.9223,E1 24.9836,E2 354.3681} C_DIS
LIN {X -13.7349,Y 111.5759,Z 120,A 92.8188,B 24.9307,C -1.9216,E1 24.9797,E2 352.9515} C_DIS
LIN {X -16.4564,Y 111.207,Z 120,A 94.2205,B 24.9308,C -1.9207,E1 24.9758,E2 351.5507} C_DIS
LIN {X -19.2157,Y 110.7638,Z 120,A 95.6468,B 24.9309,C -1.9198,E1 24.9719,E2 350.1253} C_DIS
LIN {X -21.9181,Y 110.2608,Z 120,A 97.0502,B 24.9309,C -1.9187,E1 24.968,E2 348.7228} C_DIS
LIN {X -24.5881,Y 109.6961,Z 120,A 98.4441,B 24.9311,C -1.9176,E1 24.9642,E2 347.3298} C_DIS
LIN {X -27.2598,Y 109.0628,Z 120,A 99.8395,B 24.9311,C -1.9161,E1 24.9605,E2 345.936} C_DIS
LIN {X -29.9808,Y 108.3467,Z 120,A 101.2838,B 24.9312,C -1.9151,E1 24.9566,E2 344.4921} C_DIS
LIN {X -32.6077,Y 107.5851,Z 120,A 102.681,B 24.9313,C -1.9136,E1 24.9528,E2 343.0958} C_DIS
LIN {X -35.2506,Y 106.7485,Z 120,A 104.0973,B 24.9315,C -1.9121,E1 24.9491,E2 341.6807} C_DIS
LIN {X -37.8609,Y 105.8508,Z 120,A 105.5082,B 24.9315,C -1.9105,E1 24.9453,E2 340.2709} C_DIS
LIN {X -40.4246,Y 104.8984,Z 120,A 106.9058,B 24.9317,C -1.9088,E1 24.9417,E2 338.8743} C_DIS
LIN {X -42.9372,Y 103.8949,Z 120,A 108.2881,B 24.9318,C -1.907,E1 24.9381,E2 337.4932} C_DIS
LIN {X -45.3853,Y 102.8485,Z 120,A 109.6594,B 24.9319,C -1.9056,E1 24.9346,E2 336.122} C_DIS
LIN {X -48.0328,Y 101.6399,Z 120,A 111.1372,B 24.9321,C -1.9031,E1 24.9309,E2 334.6466} C_DIS
LIN {X -50.5264,Y 100.4237,Z 120,A 112.5581,B 24.9322,C -1.9011,E1 24.9273,E2 333.2267} C_DIS
LIN {X -52.9705,Y 99.1562,Z 120,A 113.9662,B 24.9324,C -1.8989,E1 24.9239,E2 331.8199} C_DIS
LIN {X -55.3988,Y 97.8203,Z 120,A 115.3842,B 24.9326,C -1.8966,E1 24.9204,E2 330.4031} C_DIS
LIN {X -57.8062,Y 96.4172,Z 120,A 116.8038,B 24.9328,C -1.894,E1 24.917,E2 328.9855} C_DIS
LIN {X -59.762,Y 95.2153,Z 120,A 118.0354,B 24.9328,C -1.8943,E1 24.9141,E2 327.7493} C_DIS
LIN {X -62.4269,Y 93.4917,Z 120,A 119.6095,B 24.9331,C -1.8894,E1 24.9104,E2 326.1818} C_DIS
LIN {X -64.6887,Y 91.9411,Z 120,A 121.013,B 24.9333,C -1.8868,E1 24.9072,E2 324.7796} C_DIS
LIN {X -66.9086,Y 90.3383,Z 120,A 122.4146,B 24.9335,C -1.8842,E1 24.904,E2 323.3794} C_DIS
LIN {X -69.219,Y 88.5805,Z 120,A 124.0665,B 24.9332,C -1.8879,E1 24.9004,E2 321.7125} C_DIS
LIN {X -71.8925,Y 86.4225,Z 120,A 125.7531,B 24.9336,C -1.8815,E1 24.8967,E2 320.0348} C_DIS
LIN {X -74.4656,Y 84.2183,Z 120,A 127.3963,B 24.9342,C -1.8741,E1 24.8933,E2 318.4027} C_DIS
LIN {X -76.4992,Y 82.3754,Z 120,A 128.8022,B 24.9344,C -1.8712,E1 24.8904,E2 316.9982} C_DIS
LIN {X -78.7733,Y 80.2014,Z 120,A 130.5015,B 24.9344,C -1.8712,E1 24.887,E2 315.2918} C_DIS
LIN {X -80.9352,Y 78.0185,Z 120,A 131.9899,B 24.9349,C -1.8642,E1 24.8841,E2 313.8135} C_DIS
LIN {X -82.829,Y 76.0049,Z 120,A 133.4212,B 24.935,C -1.8616,E1 24.8814,E2 312.3822} C_DIS
LIN {X -84.6961,Y 73.9186,Z 120,A 134.8353,B 24.9353,C -1.8574,E1 24.8788,E2 310.9717} C_DIS
LIN {X -86.6439,Y 71.6262,Z 120,A 136.4227,B 24.9355,C -1.8555,E1 24.8759,E2 309.3815} C_DIS
LIN {X -88.5966,Y 69.1986,Z 120,A 137.9786,B 24.9358,C -1.85,E1 24.8732,E2 307.8315} C_DIS
LIN {X -90.2427,Y 67.0373,Z 120,A 139.3706,B 24.9361,C -1.8465,E1 24.8709,E2 306.4411} C_DIS
LIN {X -91.8079,Y 64.8765,Z 120,A 140.7367,B 24.9363,C -1.843,E1 24.8687,E2 305.0766} C_DIS
LIN {X -93.4641,Y 62.4684,Z 120,A 142.2385,B 24.9366,C -1.8393,E1 24.8663,E2 303.5763} C_DIS
LIN {X -94.9639,Y 60.1638,Z 120,A 143.6484,B 24.9368,C -1.8357,E1 24.8642,E2 302.1679} C_DIS
LIN {X -96.4164,Y 57.8075,Z 120,A 145.0681,B 24.9371,C -1.8319,E1 24.8622,E2 300.7498} C_DIS
LIN {X -97.587,Y 55.8052,Z 120,A 146.2947,B 24.9372,C -1.8303,E1 24.8604,E2 299.5208} C_DIS
LIN {X -99.0058,Y 53.2484,Z 120,A 147.7126,B 24.9377,C -1.823,E1 24.8586,E2 298.1126} C_DIS
LIN {X -100.2936,Y 50.7815,Z 120,A 149.2048,B 24.9377,C -1.8217,E1 24.8566,E2 296.6156} C_DIS
LIN {X -101.6189,Y 48.0774,Z 120,A 150.7309,B 24.9381,C -1.8167,E1 24.8548,E2 295.0931} C_DIS
LIN {X -102.7731,Y 45.5581,Z 120,A 152.1519,B 24.9384,C -1.8128,E1 24.8532,E2 293.6737} C_DIS
LIN {X -103.8585,Y 43.0263,Z 120,A 153.5651,B 24.9387,C -1.8088,E1 24.8516,E2 292.2622} C_DIS
LIN {X -104.852,Y 40.5439,Z 120,A 154.939,B 24.9389,C -1.805,E1 24.8502,E2 290.8896} C_DIS
LIN {X -105.8365,Y 37.9007,Z 120,A 156.3845,B 24.9392,C -1.8008,E1 24.8489,E2 289.4459} C_DIS
LIN {X -106.6576,Y 35.5207,Z 120,A 157.6937,B 24.9394,C -1.7978,E1 24.8477,E2 288.1363} C_DIS
LIN {X -107.5661,Y 32.6702,Z 120,A 159.2055,B 24.9398,C -1.7925,E1 24.8464,E2 286.6286} C_DIS
LIN {X -108.22,Y 30.428,Z 120,A 160.4624,B 24.9398,C -1.7913,E1 24.8455,E2 285.3672} C_DIS
LIN {X -109.0312,Y 27.3855,Z 120,A 162.0333,B 24.9403,C -1.7849,E1 24.8444,E2 283.8026} C_DIS
LIN {X -109.6845,Y 24.6408,Z 120,A 163.477,B 24.9406,C -1.7805,E1 24.8435,E2 282.361} C_DIS
LIN {X -110.2586,Y 21.9293,Z 120,A 164.8956,B 24.9409,C -1.7761,E1 24.8427,E2 280.9442} C_DIS
LIN {X -110.7625,Y 19.2228,Z 120,A 166.3097,B 24.9411,C -1.772,E1 24.842,E2 279.5316} C_DIS
LIN {X -111.2,Y 16.5049,Z 120,A 167.7234,B 24.9414,C -1.7679,E1 24.8414,E2 278.1193} C_DIS
LIN {X -111.5701,Y 13.7819,Z 120,A 169.129,B 24.9417,C -1.7635,E1 24.8409,E2 276.7157} C_DIS
LIN {X -111.8775,Y 11.0121,Z 120,A 170.562,B 24.942,C -1.7594,E1 24.8405,E2 275.2839} C_DIS
LIN {X -112.1121,Y 8.2888,Z 120,A 171.963,B 24.9423,C -1.7552,E1 24.8402,E2 273.8846} C_DIS
LIN {X -112.2814,Y 5.5419,Z 120,A 173.3794,B 24.9425,C -1.7512,E1 24.8399,E2 272.4693} C_DIS
LIN {X -112.3839,Y 2.7734,Z 120,A 174.8073,B 24.9428,C -1.7472,E1 24.8399,E2 271.0423} C_DIS
LIN {X -112.4176,Y 0.0823,Z 120,A 176.1667,B 24.9431,C -1.7423,E1 24.8398,E2 269.6865} C_DIS
LIN {X -112.3847,Y -2.7402,Z 120,A 177.6292,B 24.9434,C -1.7385,E1 24.8398,E2 268.2241} C_DIS
LIN {X -112.2832,Y -5.5071,Z 120,A 179.0527,B 24.9436,C -1.7344,E1 24.84,E2 266.8017} C_DIS
LIN {X -112.1162,Y -8.2329,Z 120,A -179.5457,B 24.9439,C -1.7303,E1 24.8403,E2 265.4015} C_DIS
LIN {X -111.8813,Y -10.9711,Z 120,A -178.1348,B 24.9442,C -1.7262,E1 24.8407,E2 263.9919} C_DIS
LIN {X -111.5919,Y -13.5981,Z 120,A -176.7709,B 24.9444,C -1.7226,E1 24.8411,E2 262.6285} C_DIS
LIN {X -111.2052,Y -16.4691,Z 120,A -175.2924,B 24.9447,C -1.7179,E1 24.8417,E2 261.1523} C_DIS
LIN {X -110.7659,Y -19.2032,Z 120,A -173.8713,B 24.945,C -1.7139,E1 24.8423,E2 259.7325} C_DIS
LIN {X -110.295,Y -21.7404,Z 120,A -172.5366,B 24.9452,C -1.7105,E1 24.843,E2 258.3979} C_DIS
LIN {X -109.6903,Y -24.6146,Z 120,A -171.0398,B 24.9455,C -1.7058,E1 24.8439,E2 256.9035} C_DIS
LIN {X -109.0544,Y -27.294,Z 120,A -169.6268,B 24.9457,C -1.7018,E1 24.8449,E2 255.4917} C_DIS
LIN {X -108.1196,Y -30.7826,Z 120,A -167.7023,B 24.9459,C -1.6995,E1 24.8463,E2 253.5616} C_DIS
LIN {X -107.1743,Y -33.9338,Z 120,A -166.0855,B 24.9464,C -1.692,E1 24.8476,E2 251.9534} C_DIS
LIN {X -106.3109,Y -36.5488,Z 120,A -164.67,B 24.9466,C -1.6882,E1 24.8489,E2 250.5388} C_DIS
LIN {X -105.3688,Y -39.1825,Z 120,A -163.2421,B 24.9469,C -1.6841,E1 24.8502,E2 249.1127} C_DIS
LIN {X -104.4272,Y -41.6252,Z 120,A -161.8908,B 24.9471,C -1.6808,E1 24.8516,E2 247.7615} C_DIS
LIN {X -103.3327,Y -44.2741,Z 120,A -160.4254,B 24.9473,C -1.6767,E1 24.8532,E2 246.2977} C_DIS
LIN {X -102.2306,Y -46.762,Z 120,A -159.0504,B 24.9476,C -1.6723,E1 24.8548,E2 244.9258} C_DIS
LIN {X -100.4227,Y -50.5284,Z 120,A -156.8871,B 24.9479,C -1.6676,E1 24.8574,E2 242.762} C_DIS
LIN {X -99.1549,Y -52.973,Z 120,A -155.4754,B 24.9481,C -1.664,E1 24.8593,E2 241.3512} C_DIS
LIN {X -97.8897,Y -55.2745,Z 120,A -154.1181,B 24.9483,C -1.6611,E1 24.8611,E2 239.9937} C_DIS
LIN {X -96.4259,Y -57.7919,Z 120,A -152.6367,B 24.9485,C -1.657,E1 24.8632,E2 238.5145} C_DIS
LIN {X -94.99,Y -60.1226,Z 120,A -151.2329,B 24.9488,C -1.6537,E1 24.8653,E2 237.1115} C_DIS
LIN {X -93.51,Y -62.3991,Z 120,A -149.8448,B 24.949,C -1.6503,E1 24.8674,E2 235.7245} C_DIS
LIN {X -92.141,Y -64.4012,Z 120,A -148.5576,B 24.949,C -1.6492,E1 24.8695,E2 234.4335} C_DIS
LIN {X -90.3078,Y -66.9503,Z 120,A -146.9889,B 24.9494,C -1.6439,E1 24.872,E2 232.8698} C_DIS
LIN {X -88.6191,Y -69.1701,Z 120,A -145.5641,B 24.9496,C -1.6406,E1 24.8745,E2 231.4463} C_DIS
LIN {X -86.9054,Y -71.3113,Z 120,A -144.1549,B 24.9497,C -1.6377,E1 24.877,E2 230.0373} C_DIS
LIN {X -85.1278,Y -73.4242,Z 120,A -142.7406,B 24.9499,C -1.6347,E1 24.8795,E2 228.6236} C_DIS
LIN {X -83.3113,Y -75.4788,Z 120,A -141.3379,B 24.9501,C -1.6317,E1 24.8821,E2 227.2218} C_DIS
LIN {X -81.1025,Y -77.8448,Z 120,A -139.6185,B 24.9501,C -1.6309,E1 24.8854,E2 225.4968} C_DIS
LIN {X -78.9994,Y -79.978,Z 120,A -138.1452,B 24.9505,C -1.6255,E1 24.8883,E2 224.0302} C_DIS
LIN {X -77.0105,Y -81.8948,Z 120,A -136.731,B 24.9507,C -1.6228,E1 24.8912,E2 222.6165} C_DIS
LIN {X -74.9818,Y -83.7563,Z 120,A -135.3238,B 24.9508,C -1.6202,E1 24.8941,E2 221.21} C_DIS
LIN {X -72.9153,Y -85.5613,Z 120,A -133.915,B 24.951,C -1.6179,E1 24.8971,E2 219.8012} C_DIS
LIN {X -70.7911,Y -87.327,Z 120,A -132.5251,B 24.9512,C -1.6145,E1 24.9001,E2 218.4142} C_DIS
LIN {X -68.4953,Y -89.1392,Z 120,A -130.9716,B 24.9512,C -1.6143,E1 24.9035,E2 216.8553} C_DIS
LIN {X -65.854,Y -91.1104,Z 120,A -129.3203,B 24.9514,C -1.6102,E1 24.9072,E2 215.2079} C_DIS
LIN {X -63.603,Y -92.6958,Z 120,A -127.9116,B 24.9515,C -1.6081,E1 24.9104,E2 213.7995} C_DIS
LIN {X -61.4723,Y -94.1211,Z 120,A -126.604,B 24.9517,C -1.6061,E1 24.9135,E2 212.4924} C_DIS
LIN {X -59.0207,Y -95.6784,Z 120,A -125.1155,B 24.9517,C -1.6041,E1 24.917,E2 211.0038} C_DIS
LIN {X -56.6907,Y -97.0768,Z 120,A -123.7269,B 24.9519,C -1.6022,E1 24.9204,E2 209.6155} C_DIS
LIN {X -54.6146,Y -98.2582,Z 120,A -122.4503,B 24.9519,C -1.603,E1 24.9235,E2 208.3333} C_DIS
LIN {X -51.9997,Y -99.6675,Z 120,A -120.9693,B 24.9521,C -1.5996,E1 24.9271,E2 206.8562} C_DIS
LIN {X -49.3136,Y -101.0249,Z 120,A -119.4485,B 24.9522,C -1.5972,E1 24.9309,E2 205.3373} C_DIS
LIN {X -46.0806,Y -102.5377,Z 120,A -117.5951,B 24.9522,C -1.5965,E1 24.9356,E2 203.4808} C_DIS
LIN {X -43.0876,Y -103.8327,Z 120,A -115.9593,B 24.9524,C -1.5936,E1 24.9398,E2 201.8481} C_DIS
LIN {X -40.5824,Y -104.8369,Z 120,A -114.5824,B 24.9524,C -1.5924,E1 24.9434,E2 200.4713} C_DIS
LIN {X -38.2711,Y -105.7014,Z 120,A -113.2744,B 24.9524,C -1.5934,E1 24.9468,E2 199.1582} C_DIS
LIN {X -35.2711,Y -106.7417,Z 120,A -111.7001,B 24.9526,C -1.5901,E1 24.951,E2 197.5887} C_DIS
LIN {X -32.6305,Y -107.5784,Z 120,A -110.286,B 24.9526,C -1.5892,E1 24.9548,E2 196.1743} C_DIS
LIN {X -30.0039,Y -108.3402,Z 120,A -108.8888,B 24.9527,C -1.5884,E1 24.9585,E2 194.7767} C_DIS
LIN {X -27.3415,Y -109.0425,Z 120,A -107.4836,B 24.9527,C -1.5877,E1 24.9623,E2 193.3713} C_DIS
LIN {X -24.6522,Y -109.6818,Z 120,A -106.0733,B 24.9528,C -1.587,E1 24.9662,E2 191.9606} C_DIS
LIN {X -21.9438,Y -110.2557,Z 120,A -104.6615,B 24.9528,C -1.5864,E1 24.97,E2 190.5485} C_DIS
LIN {X -19.4651,Y -110.719,Z 120,A -103.359,B 24.9528,C -1.5867,E1 24.9736,E2 189.244} C_DIS
LIN {X -16.518,Y -111.198,Z 120,A -101.8521,B 24.9528,C -1.5857,E1 24.9778,E2 187.7382} C_DIS
LIN {X -13.8259,Y -111.5644,Z 120,A -100.4665,B 24.9529,C -1.5855,E1 24.9816,E2 186.3523} C_DIS
LIN {X -11.0972,Y -111.8687,Z 120,A -99.0676,B 24.9529,C -1.5853,E1 24.9855,E2 184.9529} C_DIS
LIN {X -8.6928,Y -112.0798,Z 120,A -97.7927,B 24.9528,C -1.5872,E1 24.9891,E2 183.6729} C_DIS
LIN {X -5.5829,Y -112.2791,Z 120,A -96.249,B 24.9529,C -1.5853,E1 24.9934,E2 182.1332} C_DIS
LIN {X -2.869,Y -112.381,Z 120,A -94.8666,B 24.9529,C -1.5854,E1 24.9972,E2 180.7503} C_DIS
LIN {X -0.2374,Y -112.4168,Z 120,A -93.5397,B 24.9529,C -1.5851,E1 25.0009,E2 179.4242} C_DIS
LIN {X -0.2374,Y -112.4168,Z 120,A -93.5397,B 24.9529,C -1.5851,E1 25.0009,E2 179.4242} C_DIS
Enddeposition()
LIN {X 0.835,Y -118.3416,Z 121,A -92.9953,B 24.9584,C -1.4902,E1 25.0018,E2 179.1048} C_DIS
Startdeposition()
$VEL.CP = VEL_PRINT
LIN {X -2.3447,Y -118.324,Z 121,A -94.9752,B 24.9595,C -1.4697,E1 24.9961,E2 181.1332} C_DIS
LIN {X -5.6055,Y -118.2155,Z 121,A -96.557,B 24.9595,C -1.4694,E1 24.9917,E2 182.716} C_DIS
LIN {X -8.2029,Y -118.0627,Z 121,A -97.8506,B 24.9596,C -1.4679,E1 24.9881,E2 184.0137} C_DIS
LIN {X -11.0979,Y -117.8259,Z 121,A -99.2693,B 24.9596,C -1.4674,E1 24.9842,E2 185.4342} C_DIS
LIN {X -15.4272,Y -117.3375,Z 121,A -101.3794,B 24.9596,C -1.4677,E1 24.9783,E2 187.545} C_DIS
LIN {X -18.3021,Y -116.9236,Z 121,A -102.7863,B 24.9596,C -1.4681,E1 24.9744,E2 188.9524} C_DIS
LIN {X -21.6627,Y -116.3499,Z 121,A -104.3811,B 24.9595,C -1.4711,E1 24.9701,E2 190.5416} C_DIS
LIN {X -24.0173,Y -115.8847,Z 121,A -105.6011,B 24.9595,C -1.469,E1 24.9667,E2 191.7678} C_DIS
LIN {X -27.0557,Y -115.2138,Z 121,A -107.0305,B 24.9593,C -1.4732,E1 24.9628,E2 193.1892} C_DIS
LIN {X -29.6745,Y -114.5667,Z 121,A -108.3599,B 24.9593,C -1.4729,E1 24.9592,E2 194.5212} C_DIS
LIN {X -32.4772,Y -113.8039,Z 121,A -109.8251,B 24.9595,C -1.4712,E1 24.9553,E2 195.9928} C_DIS
LIN {X -35.2603,Y -112.9726,Z 121,A -111.2336,B 24.9595,C -1.4721,E1 24.9515,E2 197.4014} C_DIS
LIN {X -38.5003,Y -111.912,Z 121,A -112.8298,B 24.9592,C -1.4758,E1 24.9473,E2 198.9918} C_DIS
LIN {X -41.2351,Y -110.9335,Z 121,A -114.2388,B 24.9592,C -1.477,E1 24.9436,E2 200.401} C_DIS
LIN {X -43.4755,Y -110.0726,Z 121,A -115.4034,B 24.9591,C -1.478,E1 24.9406,E2 201.5655} C_DIS
LIN {X -46.6287,Y -108.7765,Z 121,A -117.0574,B 24.959,C -1.4796,E1 24.9363,E2 203.2198} C_DIS
LIN {X -48.8242,Y -107.8067,Z 121,A -118.2793,B 24.959,C -1.4783,E1 24.9332,E2 204.4476} C_DIS
LIN {X -51.91,Y -106.3576,Z 121,A -119.8769,B 24.9588,C -1.4825,E1 24.9292,E2 206.0392} C_DIS
LIN {X -54.5045,Y -105.0516,Z 121,A -121.2869,B 24.9588,C -1.4842,E1 24.9257,E2 207.4491} C_DIS
LIN {X -56.9676,Y -103.7358,Z 121,A -122.6464,B 24.9586,C -1.4857,E1 24.9223,E2 208.8089} C_DIS
LIN {X -59.5934,Y -102.2506,Z 121,A -124.1079,B 24.9586,C -1.4877,E1 24.9188,E2 210.2699} C_DIS
LIN {X -62.0849,Y -100.7573,Z 121,A -125.5187,B 24.9584,C -1.4896,E1 24.9154,E2 211.6805} C_DIS
LIN {X -65.7514,Y -98.4039,Z 121,A -127.6351,B 24.9583,C -1.4926,E1 24.9105,E2 213.7966} C_DIS
LIN {X -68.9181,Y -96.2101,Z 121,A -129.5071,B 24.9581,C -1.4955,E1 24.9062,E2 215.6682} C_DIS
LIN {X -71.2585,Y -94.4898,Z 121,A -130.9585,B 24.9581,C -1.496,E1 24.9029,E2 217.1235} C_DIS
LIN {X -73.9517,Y -92.3998,Z 121,A -132.5756,B 24.9578,C -1.5005,E1 24.8994,E2 218.736} C_DIS
LIN {X -76.1971,Y -90.5571,Z 121,A -133.9877,B 24.9577,C -1.5029,E1 24.8963,E2 220.1477} C_DIS
LIN {X -78.2711,Y -88.7693,Z 121,A -135.3052,B 24.9575,C -1.5059,E1 24.8936,E2 221.4633} C_DIS
LIN {X -80.1769,Y -87.0503,Z 121,A -136.6244,B 24.9575,C -1.5051,E1 24.8908,E2 222.7896} C_DIS
LIN {X -82.6524,Y -84.7063,Z 121,A -138.2248,B 24.9572,C -1.5107,E1 24.8876,E2 224.3834} C_DIS
LIN {X -85.2333,Y -82.1056,Z 121,A -140.0421,B 24.9572,C -1.5127,E1 24.8841,E2 226.2036} C_DIS
LIN {X -87.6911,Y -79.4786,Z 121,A -141.757,B 24.9568,C -1.5177,E1 24.8808,E2 227.9141} C_DIS
LIN {X -90.5571,Y -76.1971,Z 121,A -143.8771,B 24.9566,C -1.5222,E1 24.877,E2 230.0333} C_DIS
LIN {X -92.9875,Y -73.2081,Z 121,A -145.7521,B 24.9564,C -1.5263,E1 24.8737,E2 231.9073} C_DIS
LIN {X -95.0591,Y -70.5006,Z 121,A -147.4111,B 24.9561,C -1.5299,E1 24.8709,E2 233.5655} C_DIS
LIN {X -96.7606,Y -68.1465,Z 121,A -148.8251,B 24.956,C -1.5332,E1 24.8686,E2 234.9788} C_DIS
LIN {X -98.4039,Y -65.7514,Z 121,A -150.239,B 24.9558,C -1.5364,E1 24.8664,E2 236.3919} C_DIS
LIN {X -99.9879,Y -63.3166,Z 121,A -151.6533,B 24.9556,C -1.5398,E1 24.8643,E2 237.8054} C_DIS
LIN {X -101.2496,Y -61.2749,Z 121,A -152.8793,B 24.9556,C -1.5402,E1 24.8625,E2 239.0367} C_DIS
LIN {X -103.4364,Y -57.5067,Z 121,A -154.9437,B 24.9551,C -1.5478,E1 24.8596,E2 241.0937} C_DIS
LIN {X -104.8165,Y -54.9509,Z 121,A -156.3584,B 24.9549,C -1.5514,E1 24.8578,E2 242.5074} C_DIS
LIN {X -106.1335,Y -52.362,Z 121,A -157.7438,B 24.9546,C -1.5562,E1 24.856,E2 243.8888} C_DIS
LIN {X -107.3865,Y -49.7416,Z 121,A -159.2454,B 24.9546,C -1.5562,E1 24.8542,E2 245.3985} C_DIS
LIN {X -109.1446,Y -45.7553,Z 121,A -161.3679,B 24.9543,C -1.5618,E1 24.8519,E2 247.5194} C_DIS
LIN {X -110.4191,Y -42.5933,Z 121,A -162.9716,B 24.9539,C -1.5686,E1 24.8502,E2 249.1159} C_DIS
LIN {X -111.912,Y -38.5003,Z 121,A -165.0946,B 24.9536,C -1.5743,E1 24.8482,E2 251.2372} C_DIS
LIN {X -113.2533,Y -34.355,Z 121,A -167.2176,B 24.9532,C -1.5802,E1 24.8464,E2 253.3586} C_DIS
LIN {X -114.0623,Y -31.5653,Z 121,A -168.6332,B 24.953,C -1.5841,E1 24.8454,E2 254.773} C_DIS
LIN {X -114.8026,Y -28.7565,Z 121,A -170.0488,B 24.9527,C -1.5881,E1 24.8444,E2 256.1874} C_DIS
LIN {X -115.3602,Y -26.4221,Z 121,A -171.2188,B 24.9525,C -1.5914,E1 24.8436,E2 257.3563} C_DIS
LIN {X -116.0753,Y -23.0888,Z 121,A -172.8804,B 24.9523,C -1.5961,E1 24.8427,E2 259.0165} C_DIS
LIN {X -116.7633,Y -19.2984,Z 121,A -174.8159,B 24.9521,C -1.5991,E1 24.8418,E2 260.9563} C_DIS
LIN {X -117.2017,Y -16.4271,Z 121,A -176.2319,B 24.9518,C -1.6032,E1 24.8412,E2 262.3709} C_DIS
LIN {X -117.5845,Y -13.4181,Z 121,A -177.637,B 24.9514,C -1.6105,E1 24.8407,E2 263.767} C_DIS
LIN {X -117.913,Y -10.1541,Z 121,A -179.2519,B 24.9512,C -1.6145,E1 24.8403,E2 265.3821} C_DIS
LIN {X -118.1266,Y -7.2573,Z 121,A 179.3317,B 24.9509,C -1.6186,E1 24.84,E2 266.7972} C_DIS
LIN {X -118.3137,Y -2.9044,Z 121,A 177.102,B 24.9508,C -1.6205,E1 24.8398,E2 269.0359} C_DIS
LIN {X -118.3456,Y 0.7081,Z 121,A 175.3822,B 24.9504,C -1.6275,E1 24.8398,E2 270.7494} C_DIS
LIN {X -118.2692,Y 4.3561,Z 121,A 173.6671,B 24.9499,C -1.6353,E1 24.8399,E2 272.4562} C_DIS
LIN {X -118.0627,Y 8.2029,Z 121,A 171.7314,B 24.9497,C -1.6385,E1 24.8403,E2 274.3959} C_DIS
LIN {X -117.7982,Y 11.3973,Z 121,A 170.215,B 24.9493,C -1.645,E1 24.8406,E2 275.9059} C_DIS
LIN {X -117.3375,Y 15.4272,Z 121,A 168.1911,B 24.949,C -1.6489,E1 24.8413,E2 277.9326} C_DIS
LIN {X -116.6902,Y 19.7356,Z 121,A 166.1242,B 24.9485,C -1.6575,E1 24.8422,E2 279.9912} C_DIS
LIN {X -116.0753,Y 23.0888,Z 121,A 164.4623,B 24.9482,C -1.6624,E1 24.8431,E2 281.6515} C_DIS
LIN {X -115.4737,Y 25.9305,Z 121,A 163.0463,B 24.948,C -1.6665,E1 24.8439,E2 283.0659} C_DIS
LIN {X -114.8026,Y 28.7565,Z 121,A 161.6305,B 24.9477,C -1.6706,E1 24.8448,E2 284.4802} C_DIS
LIN {X -114.0623,Y 31.5653,Z 121,A 160.2142,B 24.9474,C -1.6747,E1 24.8459,E2 285.895} C_DIS
LIN {X -112.9726,Y 35.2603,Z 121,A 158.3365,B 24.9471,C -1.6802,E1 24.8474,E2 287.7705} C_DIS
LIN {X -112.0732,Y 38.0222,Z 121,A 156.8632,B 24.947,C -1.6818,E1 24.8487,E2 289.2483} C_DIS
LIN {X -110.5978,Y 42.1215,Z 121,A 154.797,B 24.9465,C -1.6902,E1 24.8507,E2 291.3062} C_DIS
LIN {X -109.3406,Y 45.2903,Z 121,A 153.1356,B 24.9462,C -1.6948,E1 24.8524,E2 292.9659} C_DIS
LIN {X -107.5995,Y 49.2842,Z 121,A 151.0123,B 24.9458,C -1.7007,E1 24.8548,E2 295.0869} C_DIS
LIN {X -105.9366,Y 52.7592,Z 121,A 149.0874,B 24.9456,C -1.7039,E1 24.8571,E2 297.0146} C_DIS
LIN {X -104.4816,Y 55.5867,Z 121,A 147.6091,B 24.9451,C -1.711,E1 24.859,E2 298.4838} C_DIS
LIN {X -103.2202,Y 57.8937,Z 121,A 146.247,B 24.9451,C -1.711,E1 24.8609,E2 299.8529} C_DIS
LIN {X -101.5116,Y 60.8437,Z 121,A 144.6439,B 24.9447,C -1.7178,E1 24.8632,E2 301.4483} C_DIS
LIN {X -99.4759,Y 64.1143,Z 121,A 142.7094,B 24.9445,C -1.7203,E1 24.866,E2 303.3867} C_DIS
LIN {X -97.0574,Y 67.7197,Z 121,A 140.6497,B 24.944,C -1.7279,E1 24.8693,E2 305.4384} C_DIS
LIN {X -95.3572,Y 70.0936,Z 121,A 139.1727,B 24.944,C -1.7292,E1 24.8717,E2 306.9195} C_DIS
LIN {X -93.3436,Y 72.7561,Z 121,A 137.6031,B 24.9436,C -1.7355,E1 24.8744,E2 308.4817} C_DIS
LIN {X -91.4853,Y 75.08,Z 121,A 136.1556,B 24.9433,C -1.739,E1 24.8769,E2 309.9275} C_DIS
LIN {X -89.6152,Y 77.3026,Z 121,A 134.7415,B 24.9431,C -1.7423,E1 24.8794,E2 311.3401} C_DIS
LIN {X -86.7092,Y 80.5487,Z 121,A 132.6206,B 24.9428,C -1.7472,E1 24.8834,E2 313.4588} C_DIS
LIN {X -84.7063,Y 82.6524,Z 121,A 131.2065,B 24.9426,C -1.7504,E1 24.8862,E2 314.8714} C_DIS
LIN {X -81.97,Y 85.3641,Z 121,A 129.3317,B 24.9423,C -1.7545,E1 24.8899,E2 316.7442} C_DIS
LIN {X -79.8825,Y 87.3205,Z 121,A 127.9328,B 24.9421,C -1.7572,E1 24.8928,E2 318.1425} C_DIS
LIN {X -77.6826,Y 89.2833,Z 121,A 126.5051,B 24.9419,C -1.7605,E1 24.8957,E2 319.568} C_DIS
LIN {X -75.4681,Y 91.1628,Z 121,A 125.0924,B 24.9417,C -1.7633,E1 24.8988,E2 320.9793} C_DIS
LIN {X -72.8123,Y 93.3003,Z 121,A 123.4339,B 24.9415,C -1.7666,E1 24.9024,E2 322.6363} C_DIS
LIN {X -70.5006,Y 95.0591,Z 121,A 122.0215,B 24.9413,C -1.7693,E1 24.9055,E2 324.0473} C_DIS
LIN {X -68.1465,Y 96.7606,Z 121,A 120.6089,B 24.9412,C -1.7719,E1 24.9087,E2 325.4585} C_DIS
LIN {X -65.7514,Y 98.4039,Z 121,A 119.1966,B 24.941,C -1.7744,E1 24.912,E2 326.8696} C_DIS
LIN {X -62.5128,Y 100.49,Z 121,A 117.2665,B 24.941,C -1.7753,E1 24.9166,E2 328.8038} C_DIS
LIN {X -59.5934,Y 102.2506,Z 121,A 115.6667,B 24.9406,C -1.7804,E1 24.9204,E2 330.3962} C_DIS
LIN {X -56.233,Y 104.1343,Z 121,A 113.7946,B 24.9404,C -1.7834,E1 24.925,E2 332.2666} C_DIS
LIN {X -53.6605,Y 105.4829,Z 121,A 112.3833,B 24.9402,C -1.7856,E1 24.9284,E2 333.6767} C_DIS
LIN {X -51.0556,Y 106.7681,Z 121,A 110.9722,B 24.9402,C -1.7876,E1 24.932,E2 335.0866} C_DIS
LIN {X -48.42,Y 107.9889,Z 121,A 109.5612,B 24.94,C -1.7895,E1 24.9356,E2 336.4964} C_DIS
LIN {X -45.7553,Y 109.1446,Z 121,A 108.106,B 24.94,C -1.7895,E1 24.9393,E2 337.9551} C_DIS
LIN {X -42.5933,Y 110.4191,Z 121,A 106.4953,B 24.9397,C -1.7934,E1 24.9435,E2 339.5599} C_DIS
LIN {X -38.5003,Y 111.912,Z 121,A 104.3802,B 24.9395,C -1.7959,E1 24.949,E2 341.6735} C_DIS
LIN {X -34.355,Y 113.2533,Z 121,A 102.2656,B 24.9394,C -1.7981,E1 24.9547,E2 343.7864} C_DIS
LIN {X -31.5653,Y 114.0623,Z 121,A 100.8561,B 24.9394,C -1.7995,E1 24.9585,E2 345.1949} C_DIS
LIN {X -28.7565,Y 114.8026,Z 121,A 99.4468,B 24.9392,C -1.8008,E1 24.9623,E2 346.6032} C_DIS
LIN {X -25.0044,Y 115.6757,Z 121,A 97.5208,B 24.9392,C -1.7999,E1 24.9675,E2 348.534} C_DIS
Enddeposition()
END
